# B&R Automation Studio project A2019059_Linka_Power_CP (part 41)

#### Main.st - Init, cyclic, exit code
```iecst
PROGRAM _INIT
    Triger_0:= FALSE;
    Triger_1:= FALSE;

    P4_FunkcnyTestA.STAV.Tester_ON:= TRUE;
    P4_FunkcnyTestA.OUT.HorneKontakty_ZASUN_YV177:= TRUE;
END_PROGRAM

PROGRAM _CYCLIC

	//Volanie podprogramov//
    OvlCentrovacky;
    IOLinkKomunikacia;
    OvlHornychKontaktov;
    OvlSpodnychKontaktov;
    OvlTestera;

    //Volanie funkcie SequenceControl//
    SequenceControl(SC:= SC_P4_FunkcnyTestA);

    //Príznak funkčný test A východzia pozícia//
    IF P4_FunkcnyTestA.IN.Centrovanie_ZASUNUTE_MS27 AND P4_FunkcnyTestA.IN.HorneKontakty_ZASUNUTE_MS23 AND P4_FunkcnyTestA.IN.SpodneKontakty_ZASUNUTE_MS31 THEN
        P4_FunkcnyTestA_VychodziaPozicia:= TRUE;
    ELSE
        P4_FunkcnyTestA_VychodziaPozicia:= FALSE;
    END_IF

    //Reset sekcie //
    IF NOT Safety.STAV.P4_ZonaBunky_AKTIVNA THEN
        SC_P4_FunkcnyTestA.Step:= 0;
    ELSIF P4_FunkcnyTestA.Reset THEN
        SC_P4_FunkcnyTestA.Step:= 0;
        P4_FunkcnyTestA.Reset:= FALSE;
    END_IF

    //Porucha stanice//
    IF P4_PoruchaST1 AND NOT Triger_0 THEN
        Triger_0:= TRUE;
        SC_P4_FunkcnyTestA.Step:= 0;
    END_IF

    IF NOT P4_PoruchaST1 THEN
        Triger_0:= FALSE;
    END_IF

    //Čas testovania//
    CasTestovania.PT:= T#5M;
    CasTestovania();
    NameranyCasTestovania;

    CASE SC_P4_FunkcnyTestA.Step OF

        0:
            SC_P4_FunkcnyTestA.StepName:='0 - Nulovanie';
            SC_OvlCentrovacky.Step:= 0;
            SC_OvlHornychKontaktov.Step:= 0;
            SC_OvlSpodnychKontaktov.Step:= 0;
            P4_FunkcnyTestA.Automat:= FALSE;
            P4_FunkcnyTestA.KoniecCyklu:= FALSE;
            P4_FunkcnyTestA.Manual:= FALSE;
            P4_FunkcnyTestA.STAV.PoINIT:= FALSE;
            P4_FunkcnyTestA.OUT.KontaktyTestera_VYSUN_YV171:= FALSE;
            P4_FunkcnyTestA.OUT.OdpruzenieKontaktov_VYPNI_YV180:= TRUE;
            P4_FunkcnyTestA.OUT.OdpruzenieKontaktov_ZAPNI_YV179:= FALSE;
            P4_FunkcnyTestA.OUT.ZasunStoper_YV163:= FALSE;
            PrecitaneCisloPaletky:= '';
            FV_Test_START:= FALSE;
            FV_Test_UKONCENY:= FALSE;
            Taktime_FunkcnyTestA.CMD.START_Merania_1:= FALSE;
            Taktime_FunkcnyTestA.CMD.START_Merania_2:= FALSE;
            PaletkaPrechadza:= FALSE;
            P4_FunkcnyTestA.STAV.PrebiehaVyvezeniePaletky:= FALSE;
            P4_FunkcnyTestA_ZATVOR:= FALSE;
            P4_FunkcnyTestA_OTVOR:= FALSE;
            TestovaciKus:= FALSE;
            Revork:= FALSE;
            CasTestovania.IN:= FALSE;
            P4_FunkcnyTestA.RR_TestovanieFunkcnehoTestu:= FALSE;
            P4_FunkcnyTestA.RR_VysunKontaktyTestera:= FALSE;
            P4_FunkcnyTestA.RR_ZapniOdpruzenieKontaktov:= FALSE;
            P4_FunkcnyTestA.RR_OtvorTester:= FALSE;
            P4_FunkcnyTestA.RR_ZatvorTester:= FALSE;
            PocetOpakovaniTestu:= 0;
            OpakovanyTest:= FALSE;

            IF Safety.STAV.P4_ZonaBunky_AKTIVNA AND NOT P4_Pracovisko.STAV.PORUCHA AND P4_Pracovisko.IN.PrivodVzduchu_SnimacTlaku_S15 THEN
                SC_P4_FunkcnyTestA.ResetStep:= TRUE;
                SC_P4_FunkcnyTestA.Step:= 1;
            END_IF

        1:
            SC_P4_FunkcnyTestA.StepName:='1 - Cakam na spustenie vyroby';
            P4_FunkcnyTestA.KoniecCyklu:= FALSE;
            IF P4_FunkcnyTestA.Automat THEN
                SC_P4_FunkcnyTestA.Step:= 2;
            ELSIF P4_FunkcnyTestA.Manual THEN
                SC_P4_FunkcnyTestA.Step:= 700;
            ELSIF P4_FunkcnyTestA_ZATVOR THEN
                SC_P4_FunkcnyTestA.Step:= 720;
            ELSIF P4_FunkcnyTestA_OTVOR THEN
                SC_P4_FunkcnyTestA.Step:= 750;
            END_IF

            //********************************************************Inicializácia****************************************************************************//

        2:
            SC_P4_FunkcnyTestA.StepName:='2 - Inicializacia - cakam na spustenie inicializacie';
            SC_P4_FunkcnyTestA.IdleTime.PT:= T#2s;
            SC_P4_FunkcnyTestA.AlarmTime.PT:= T#5s;

            SC_P4_FunkcnyTestA.IdleTime.IN:= TRUE;

            IF SC_P4_FunkcnyTestA.IdleTime.Q THEN
                SC_P4_FunkcnyTestA.ResetStep:= TRUE;
                SC_P4_FunkcnyTestA.Step:= 3;
            END_IF

        3:
            SC_P4_FunkcnyTestA.StepName:='3 - Inicializacia - zasunutie hornych kontaktov';
            SC_P4_FunkcnyTestA.IdleTime.PT:= T#2s;
            SC_P4_FunkcnyTestA.AlarmTime.PT:= T#5s;

            IF NOT SC_P4_FunkcnyTestA.Switch1 THEN
                HorneKontakty_ZASUN:= TRUE;
                SC_P4_FunkcnyTestA.Switch1:= TRUE;
            END_IF

            IF P4_FunkcnyTestA.IN.HorneKontakty_ZASUNUTE_MS23 THEN
                SC_P4_FunkcnyTestA.ResetStep:= TRUE;
                SC_P4_FunkcnyTestA.Step:= 5;
            END_IF

        5:
            SC_P4_FunkcnyTestA.StepName:='5 - Inicializacia - zasunutie spodnych kontaktov';
            SC_P4_FunkcnyTestA.IdleTime.PT:= T#2s;
            SC_P4_FunkcnyTestA.AlarmTime.PT:= T#5s;

            IF NOT SC_P4_FunkcnyTestA.Switch1 THEN
                SpodneKontakty_ZASUN:= TRUE;
                SC_P4_FunkcnyTestA.Switch1:= TRUE;
            END_IF

            IF P4_FunkcnyTestA.IN.SpodneKontakty_ZASUNUTE_MS31 THEN
                SC_P4_FunkcnyTestA.ResetStep:= TRUE;
                SC_P4_FunkcnyTestA.Step:= 8;
            END_IF

        8:
            SC_P4_FunkcnyTestA.StepName:='8 - Inicializacia - zasunutie centrovacky';
            SC_P4_FunkcnyTestA.IdleTime.PT:= T#4s;
            SC_P4_FunkcnyTestA.AlarmTime.PT:= T#5s;

            IF NOT SC_P4_FunkcnyTestA.Switch1 THEN
                Centrovacku_ZASUN:= TRUE;
                SC_P4_FunkcnyTestA.Switch1:= TRUE;
            END_IF

            IF P4_FunkcnyTestA.IN.Centrovanie_ZASUNUTE_MS27 AND P4_Dopravniky.STAV.PoINIT THEN
                SC_P4_FunkcnyTestA.ResetStep:= TRUE;
                SC_P4_FunkcnyTestA.Step:= 10;
            END_IF

        10:
            SC_P4_FunkcnyTestA.StepName:='10 - Inicializacia - kontrola kontaktov funkcneho testu';
            SC_P4_FunkcnyTestA.IdleTime.PT:= T#4s;
            SC_P4_FunkcnyTestA.AlarmTime.PT:= T#5s;

            IF Linka.PAR.ZvolenyModel = '4F' AND P4_FunkcnyTestA.IN.TypSpodnychKontaktov_4F THEN
                SC_P4_FunkcnyTestA.ResetStep:= TRUE;
                SC_P4_FunkcnyTestA.Step:= 13;
            ELSIF Linka.PAR.ZvolenyModel = '5F' AND P4_FunkcnyTestA.IN.TypSpodnychKontaktov_5F_5H THEN
                SC_P4_FunkcnyTestA.ResetStep:= TRUE;
                SC_P4_FunkcnyTestA.Step:= 13;
            ELSIF Linka.PAR.ZvolenyModel = '5H'AND P4_FunkcnyTestA.IN.TypSpodnychKontaktov_5F_5H THEN
                SC_P4_FunkcnyTestA.ResetStep:= TRUE;
                SC_P4_FunkcnyTestA.Step:= 13;
            ELSE
                P34_Alarmy[437]:= TRUE;
                P4_PoruchaST1:= TRUE;
            END_IF

        13:
            SC_P4_FunkcnyTestA.StepName:='13 - Inicializacia - hladanie paletky';
            SC_P4_FunkcnyTestA.IdleTime.PT:= T#5s;
            SC_P4_FunkcnyTestA.AlarmTime.PT:= T#5s;
            SC_P4_FunkcnyTestA.IdleTime.IN:= TRUE;

            IF P4_FunkcnyTestA.IN.PritomnostPaletky_S10 THEN
                P3_LeakageTestB.STAV.PrebiehaVyvezeniePaletky:= FALSE;
                SC_P4_FunkcnyTestA.ResetStep:= TRUE;
                SC_P4_FunkcnyTestA.Step:= 20;
            ELSIF SC_P4_FunkcnyTestA.IdleTime.Q THEN
                P4_FunkcnyTestA.STAV.PoINIT:= TRUE;
                SC_P4_FunkcnyTestA.ResetStep:= TRUE;
                SC_P4_FunkcnyTestA.Step:= 100;
            END_IF

        20:
            SC_P4_FunkcnyTestA.StepName:='20 - Inicializacia - precitanie cisla paletky';
            SC_P4_FunkcnyTestA.IdleTime.PT:= T#200ms;
            SC_P4_FunkcnyTestA.AlarmTime.PT:= T#5s;
            SC_P4_FunkcnyTestA.IdleTime.IN:= TRUE;

            IF SC_P4_FunkcnyTestA.IdleTime.Q THEN
                PrecitaneCisloPaletky:= USINT_TO_STRING(P4_FunkcnyTestA.IN.PrecitaneCisloPaletky_S10);
                i:= 0;
                SC_P4_FunkcnyTestA.ResetStep:= TRUE;
                SC_P4_FunkcnyTestA.Step:= 23;
            END_IF

        23:
            SC_P4_FunkcnyTestA.StepName:='23 - Inicializacia - priradenie indexu paletky na zaklade precitanej hodnoty';
            SC_P4_FunkcnyTestA.IdleTime.PT:= T#200ms;
            SC_P4_FunkcnyTestA.AlarmTime.PT:= T#5s;

            IF PrecitaneCisloPaletky = '171' THEN
                i:= 1;
            ELSIF PrecitaneCisloPaletky = '164' THEN
                i:= 2;
            ELSIF PrecitaneCisloPaletky = '181' THEN
                i:= 3;
            ELSIF PrecitaneCisloPaletky = '168' THEN
                i:= 4;
            ELSIF PrecitaneCisloPaletky = '140' THEN
                i:= 5;
            ELSIF PrecitaneCisloPaletky = '110' THEN
                i:= 6;
            ELSIF PrecitaneCisloPaletky = '156' THEN
                i:= 7;
            ELSIF PrecitaneCisloPaletky = '127' THEN
                i:= 8;
            ELSIF PrecitaneCisloPaletky = '139' THEN
                i:= 9;
            ELSIF PrecitaneCisloPaletky = '131' THEN
                i:= 10;
            ELSIF PrecitaneCisloPaletky = '178' THEN
                i:= 11;
            ELSIF PrecitaneCisloPaletky = '206' THEN
                i:= 12;
            ELSIF PrecitaneCisloPaletky = '119' THEN
                i:= 13;
            ELSIF PrecitaneCisloPaletky = '163' THEN
                i:= 14;
            ELSIF PrecitaneCisloPaletky = '128' THEN
                i:= 15;
            ELSIF PrecitaneCisloPaletky = '175' THEN
                i:= 16;
            ELSIF PrecitaneCisloPaletky = '138' THEN
                i:= 17;
            ELSE
                P34_Alarmy[427]:= TRUE;
                P4_PoruchaST1:= TRUE;
            END_IF

            IF i<> 0 THEN
                Paletka[i].PAR.CisloPaletky:= USINT_TO_STRING(i);
                PrecitaneCisloPaletky:= '';
                SC_P4_FunkcnyTestA.ResetStep:= TRUE;
                SC_P4_FunkcnyTestA.Step:= 30;
            END_IF

        30:
            SC_P4_FunkcnyTestA.StepName:='30 - Inicializacia - kontrola stavu paletky';
            SC_P4_FunkcnyTestA.IdleTime.PT:= T#200ms;
            SC_P4_FunkcnyTestA.AlarmTime.PT:= T#5s;

            IF Paletka[i].PAR.TestovaciKus AND Paletka[i].PAR.CisloTestovacejStanice = 'ST_FT1,FT2' THEN
                IF P4_FunkcnyTestA.STAV.Tester_ON THEN
                    TestovaciKus:= TRUE;
                    P4_FunkcnyTestA.STAV.PoINIT:= TRUE;
                    SC_P4_FunkcnyTestA.ResetStep:= TRUE;
                    SC_P4_FunkcnyTestA.Step:= 118;
                ELSE
                    P4_FunkcnyTestA.STAV.PoINIT:= TRUE;
                    SC_P4_FunkcnyTestA.ResetStep:= TRUE;
                    SC_P4_FunkcnyTestA.Step:= 560;
                END_IF
            ELSIF Paletka[i].PAR.TestovaciKus AND Paletka[i].PAR.CisloTestovacejStanice <> 'ST_FT1,FT2' THEN
                P4_FunkcnyTestA.STAV.PoINIT:= TRUE;
                SC_P4_FunkcnyTestA.ResetStep:= TRUE;
                SC_P4_FunkcnyTestA.Step:= 560;
            ELSIF Paletka[i].PAR.RevorkovyKus AND Paletka[i].PAR.CisloRevorkovejStanice = 'ST_FT1,FT2' THEN
                IF P4_FunkcnyTestA.STAV.Tester_ON THEN
                    Revork:= TRUE;
                    P4_FunkcnyTestA.STAV.PoINIT:= TRUE;
                    SC_P4_FunkcnyTestA.ResetStep:= TRUE;
                    SC_P4_FunkcnyTestA.Step:= 105;
                ELSE
                    P4_FunkcnyTestA.STAV.PoINIT:= TRUE;
                    SC_P4_FunkcnyTestA.ResetStep:= TRUE;
                    SC_P4_FunkcnyTestA.Step:= 560;
                END_IF
            ELSIF Paletka[i].PAR.RevorkovyKus AND Paletka[i].PAR.CisloRevorkovejStanice <> 'ST_FT1,FT2' THEN
                Revork:= FALSE;
                P4_FunkcnyTestA.STAV.PoINIT:= TRUE;
                SC_P4_FunkcnyTestA.ResetStep:= TRUE;
                SC_P4_FunkcnyTestA.Step:= 560;
            ELSIF Paletka[i].PAR.StavPaletky = 'OK' THEN
                SC_P4_FunkcnyTestA.ResetStep:= TRUE;
                SC_P4_FunkcnyTestA.Step:= 33;
            ELSIF Paletka[i].PAR.StavPaletky = 'NG' THEN
                P4_FunkcnyTestA.STAV.PoINIT:= TRUE;
                SC_P4_FunkcnyTestA.ResetStep:= TRUE;
                SC_P4_FunkcnyTestA.Step:= 560;
            END_IF

        33:
            SC_P4_FunkcnyTestA.StepName:='33 - Inicializacia - kontrola ukoncenia testu';
            SC_P4_FunkcnyTestA.IdleTime.PT:= T#200ms;
            SC_P4_FunkcnyTestA.AlarmTime.PT:= T#5s;

            IF Paletka[i].VnutornyStav.FunkcnyTest_Ukonceny THEN
                P4_FunkcnyTestA.STAV.PoINIT:= TRUE;
                SC_P4_FunkcnyTestA.ResetStep:= TRUE;
                SC_P4_FunkcnyTestA.Step:= 560;
            ELSE
                P4_FunkcnyTestA.STAV.PoINIT:= TRUE;
                SC_P4_FunkcnyTestA.ResetStep:= TRUE;
                SC_P4_FunkcnyTestA.Step:= 100;
            END_IF

            //********************************************************Automatický režim****************************************************************************//

        100:
            SC_P4_FunkcnyTestA.StepName:='100 - Automaticky Rezim - cakam na príchod paletky na stoper';
            SC_P4_FunkcnyTestA.IdleTime.PT:= T#200ms;
            SC_P4_FunkcnyTestA.AlarmTime.PT:= T#5s;

            IF P4_FunkcnyTestA.IN.PritomnostPaletky_S10 THEN
                P3_LeakageTestB.STAV.PrebiehaVyvezeniePaletky:= FALSE;
            END_IF

            SC_P4_FunkcnyTestA.IdleTime.IN:= P4_FunkcnyTestA.IN.PritomnostPaletky_S10;

            IF EDGEPOS(P4_FunkcnyTestA.IN.PritomnostPaletky_S10)THEN
                IF NOT Taktime_FunkcnyTestA.CMD.START_Merania_1 THEN
                    Taktime_FunkcnyTestA.CMD.START_Merania_1:= TRUE;
                ELSE
                    Taktime_FunkcnyTestA.CMD.ZAPIS_Hodnot_1:= TRUE;
                END_IF
            END_IF

            IF P4_FunkcnyTestA.KoniecCyklu THEN
                SC_P4_FunkcnyTestA.ResetStep:= TRUE;
                SC_P4_FunkcnyTestA.Step:= 0;
            ELSIF SC_P4_FunkcnyTestA.IdleTime.Q THEN
                SC_P4_FunkcnyTestA.ResetStep:= TRUE;
                SC_P4_FunkcnyTestA.Step:= 101;
            END_IF

        101:
            SC_P4_FunkcnyTestA.StepName:='101 - Automaticky Rezim - precitanie cisla paletky';
            SC_P4_FunkcnyTestA.IdleTime.PT:= T#500ms;
            SC_P4_FunkcnyTestA.AlarmTime.PT:= T#5s;
            SC_P4_FunkcnyTestA.IdleTime.IN:= TRUE;

            PrecitaneCisloPaletky:= USINT_TO_STRING(P4_FunkcnyTestA.IN.PrecitaneCisloPaletky_S10);
            i:= 0;
            SC_P4_FunkcnyTestA.ResetStep:= TRUE;
            SC_P4_FunkcnyTestA.Step:= 102;

        102:
            SC_P4_FunkcnyTestA.StepName:='102 - Automaticky Rezim - priradenie indexu paletky na zaklade precitanej hodnoty';
            SC_P4_FunkcnyTestA.IdleTime.PT:= T#200ms;
            SC_P4_FunkcnyTestA.AlarmTime.PT:= T#5s;

            IF PrecitaneCisloPaletky = '171' THEN
                i:= 1;
            ELSIF PrecitaneCisloPaletky = '164' THEN
                i:= 2;
            ELSIF PrecitaneCisloPaletky = '181' THEN
                i:= 3;
            ELSIF PrecitaneCisloPaletky = '168' THEN
                i:= 4;
            ELSIF PrecitaneCisloPaletky = '140' THEN
                i:= 5;
            ELSIF PrecitaneCisloPaletky = '110' THEN
                i:= 6;
            ELSIF PrecitaneCisloPaletky = '156' THEN
                i:= 7;
            ELSIF PrecitaneCisloPaletky = '127' THEN
                i:= 8;
            ELSIF PrecitaneCisloPaletky = '139' THEN
                i:= 9;
            ELSIF PrecitaneCisloPaletky = '131' THEN
                i:= 10;
            ELSIF PrecitaneCisloPaletky = '178' THEN
                i:= 11;
            ELSIF PrecitaneCisloPaletky = '206' THEN
                i:= 12;
            ELSIF PrecitaneCisloPaletky = '119' THEN
                i:= 13;
            ELSIF PrecitaneCisloPaletky = '163' THEN
                i:= 14;
            ELSIF PrecitaneCisloPaletky = '128' THEN
                i:= 15;
            ELSIF PrecitaneCisloPaletky = '175' THEN
                i:= 16;
            ELSIF PrecitaneCisloPaletky = '138' THEN
                i:= 17;
            ELSE
                P34_Alarmy[427]:= TRUE;
                P4_PoruchaST1:= TRUE;
            END_IF

            IF i<> 0 THEN
                Paletka[i].PAR.CisloPaletky:= USINT_TO_STRING(i);
                PrecitaneCisloPaletky:= '';
                SC_P4_FunkcnyTestA.ResetStep:= TRUE;
                SC_P4_FunkcnyTestA.Step:= 103;
            END_IF

        103:
            SC_P4_FunkcnyTestA.StepName:='108 - Automaticky Rezim - kontrola stavu paletky';
            SC_P4_FunkcnyTestA.IdleTime.PT:= T#200ms;
            SC_P4_FunkcnyTestA.AlarmTime.PT:= T#5s;

            IF Paletka[i].PAR.TestovaciKus AND Paletka[i].PAR.CisloTestovacejStanice = 'ST_FT1,FT2' THEN
                IF P4_FunkcnyTestA.STAV.Tester_ON THEN
                    TestovaciKus:= TRUE;
                    SC_P4_FunkcnyTestA.ResetStep:= TRUE;
                    SC_P4_FunkcnyTestA.Step:= 118;
                ELSE
                    SC_P4_FunkcnyTestA.ResetStep:= TRUE;
                    SC_P4_FunkcnyTestA.Step:= 560;
                END_IF
            ELSIF Paletka[i].PAR.TestovaciKus AND Paletka[i].PAR.CisloTestovacejStanice <> 'ST_FT1,FT2' THEN
                SC_P4_FunkcnyTestA.ResetStep:= TRUE;
                SC_P4_FunkcnyTestA.Step:= 560;
            ELSIF Paletka[i].PAR.RevorkovyKus AND Paletka[i].PAR.CisloRevorkovejStanice = 'ST_FT1,FT2' THEN
                IF P4_FunkcnyTestA.STAV.Tester_ON THEN
                    Revork:= TRUE;
                    SC_P4_FunkcnyTestA.ResetStep:= TRUE;
                    SC_P4_FunkcnyTestA.Step:= 105;
                ELSE
                    SC_P4_FunkcnyTestA.ResetStep:= TRUE;
                    SC_P4_FunkcnyTestA.Step:= 560;
                END_IF
            ELSIF Paletka[i].PAR.RevorkovyKus AND Paletka[i].PAR.CisloRevorkovejStanice <> 'ST_FT1,FT2' THEN
                Revork:= FALSE;
                SC_P4_FunkcnyTestA.ResetStep:= TRUE;
                SC_P4_FunkcnyTestA.Step:= 560;
            ELSIF Paletka[i].PAR.StavPaletky = 'OK' AND P4_FunkcnyTestA.STAV.Tester_ON THEN
                SC_P4_FunkcnyTestA.ResetStep:= TRUE;
                SC_P4_FunkcnyTestA.Step:= 105;
            ELSIF Paletka[i].PAR.StavPaletky = 'OK' AND NOT P4_FunkcnyTestA.STAV.Tester_ON THEN
                SC_P4_FunkcnyTestA.ResetStep:= TRUE;
                SC_P4_FunkcnyTestA.Step:= 560;
            ELSIF Paletka[i].PAR.StavPaletky = 'NG' THEN
                SC_P4_FunkcnyTestA.ResetStep:= TRUE;
                SC_P4_FunkcnyTestA.Step:= 560;
            END_IF

        105:
            SC_P4_FunkcnyTestA.StepName:='105 - Automaticky Rezim - kontrola zapnutia testovacej stanice B';
            SC_P4_FunkcnyTestA.IdleTime.PT:= T#200ms;
            SC_P4_FunkcnyTestA.AlarmTime.PT:= T#5s;

            IF P4_FunkcnyTestB.STAV.Tester_ON THEN
                SC_P4_FunkcnyTestA.ResetStep:= TRUE;
                SC_P4_FunkcnyTestA.Step:= 107;
            ELSE
                SC_P4_FunkcnyTestA.ResetStep:= TRUE;
                SC_P4_FunkcnyTestA.Step:= 118;
            END_IF

        107:
            SC_P4_FunkcnyTestA.StepName:='107 - Automaticky Rezim - kontrola paletky v testovacej stanici B';
            SC_P4_FunkcnyTestA.IdleTime.PT:= T#1s;
            SC_P4_FunkcnyTestA.AlarmTime.PT:= T#5s;
            SC_P4_FunkcnyTestA.IdleTime.IN:= TRUE;

            IF P4_FunkcnyTestA.KoniecCyklu THEN
                SC_P4_FunkcnyTestA.ResetStep:= TRUE;
                SC_P4_FunkcnyTestA.Step:= 118;
            ELSIF SC_P4_FunkcnyTestB.Step = 100 AND NOT P4_FunkcnyTestB.IN.PritomnostPaletky_S11 THEN
                SC_P4_FunkcnyTestA.ResetStep:= TRUE;
                SC_P4_FunkcnyTestA.Step:= 560;
            ELSIF SC_P4_FunkcnyTestB.Step = 110 AND P4_FunkcnyTestB.IN.PritomnostPaletky_S11 THEN
                SC_P4_FunkcnyTestA.ResetStep:= TRUE;
                SC_P4_FunkcnyTestA.Step:= 110;
            END_IF

        110:
            SC_P4_FunkcnyTestA.StepName:='110 - Automaticky Rezim - cakam na spustenie testovania';
            SC_P4_FunkcnyTestA.IdleTime.PT:= T#200ms;
            SC_P4_FunkcnyTestA.AlarmTime.PT:= T#5s;

            IF P4_FunkcnyTestB.OUT.KOM_StanicaA_StartTestovania THEN
                P4_FunkcnyTestB.OUT.KOM_StanicaA_StartTestovania:= FALSE;
                SC_P4_FunkcnyTestA.ResetStep:= TRUE;
                SC_P4_FunkcnyTestA.Step:= 118;
            END_IF

        118:
            SC_P4_FunkcnyTestA.StepName:='118 - Automaticky Rezim - zacentrovanie paletky';
            SC_P4_FunkcnyTestA.IdleTime.PT:= T#200ms;
            SC_P4_FunkcnyTestA.AlarmTime.PT:= T#5s;

            IF NOT SC_P4_FunkcnyTestA.Switch1 THEN
                Centrovacku_VYSUN:= TRUE;
                SC_P4_FunkcnyTestA.Switch1:= TRUE;
            END_IF

            IF P4_FunkcnyTestA.IN.Centrovanie_VYSUNUTE_MS29 THEN
                SC_P4_FunkcnyTestA.ResetStep:= TRUE;
                SC_P4_FunkcnyTestA.Step:= 120;
            END_IF

        120:
            SC_P4_FunkcnyTestA.StepName:='120 - Automaticky Rezim - zapnutie pruzenia vrchnych kontaktov';
            SC_P4_FunkcnyTestA.IdleTime.PT:= T#200ms;
            SC_P4_FunkcnyTestA.AlarmTime.PT:= T#5s;

            IF NOT SC_P4_FunkcnyTestA.Switch1 THEN
                P4_FunkcnyTestA.OUT.OdpruzenieKontaktov_VYPNI_YV180:= FALSE;
                P4_FunkcnyTestA.OUT.OdpruzenieKontaktov_ZAPNI_YV179:= TRUE;
                SC_P4_FunkcnyTestA.IdleTime.IN:= TRUE;
                SC_P4_FunkcnyTestA.Switch1:= TRUE;
            END_IF

            IF SC_P4_FunkcnyTestA.IdleTime.Q THEN
                SC_P4_FunkcnyTestA.ResetStep:= TRUE;
                SC_P4_FunkcnyTestA.Step:= 123;
            END_IF

        123:
            SC_P4_FunkcnyTestA.StepName:='123 - Automaticky Rezim - vysunutie hornych kontaktov';
            SC_P4_FunkcnyTestA.IdleTime.PT:= T#200ms;
            SC_P4_FunkcnyTestA.AlarmTime.PT:= T#5s;

            IF NOT SC_P4_FunkcnyTestA.Switch1 THEN
                HorneKontakty_VYSUN:= TRUE;
                SC_P4_FunkcnyTestA.Switch1:= TRUE;
            END_IF

            IF P4_FunkcnyTestA.IN.HorneKontakty_VYSUNUTE_MS25 THEN
                SC_P4_FunkcnyTestA.ResetStep:= TRUE;
                SC_P4_FunkcnyTestA.Step:= 125;
            END_IF

        125:
            SC_P4_FunkcnyTestA.StepName:='125 - Automaticky Rezim - vysunutie spodnych kontaktov';
            SC_P4_FunkcnyTestA.IdleTime.PT:= T#200ms;
            SC_P4_FunkcnyTestA.AlarmTime.PT:= T#5s;

            IF NOT SC_P4_FunkcnyTestA.Switch1 THEN
                SpodneKontakty_VYSUN:= TRUE;
                SC_P4_FunkcnyTestA.Switch1:= TRUE;
            END_IF

            IF P4_FunkcnyTestA.IN.SpodneKontakty_VYSUNUTE_MS33 THEN
                SC_P4_FunkcnyTestA.ResetStep:= TRUE;
                SC_P4_FunkcnyTestA.Step:= 127;
            END_IF

        127:
            SC_P4_FunkcnyTestA.StepName:='127 - Automaticky Rezim - pritlacenie kontaktov';
            SC_P4_FunkcnyTestA.IdleTime.PT:= T#200ms;
            SC_P4_FunkcnyTestA.AlarmTime.PT:= T#5s;

            IF Linka.PAR.ZvolenyModel = '4F' THEN
                P4_FunkcnyTestA.OUT.KontaktyTestera_VYSUN_YV171:= TRUE;
                SC_P4_FunkcnyTestA.IdleTime.IN:= TRUE;
            ELSIF Linka.PAR.ZvolenyModel = '5F' THEN
                P4_FunkcnyTestA.OUT.KontaktyTestera_VYSUN_YV171:= TRUE;
                SC_P4_FunkcnyTestA.IdleTime.IN:= TRUE;
            ELSIF Linka.PAR.ZvolenyModel = '5H' THEN
                SC_P4_FunkcnyTestA.ResetStep:= TRUE;
                SC_P4_FunkcnyTestA.Step:= 130;
            END_IF

            IF SC_P4_FunkcnyTestA.IdleTime.Q THEN
                SC_P4_FunkcnyTestA.ResetStep:= TRUE;
                SC_P4_FunkcnyTestA.Step:= 130;
            END_IF

        130:
            SC_P4_FunkcnyTestA.StepName:='130 - Automaticky Rezim - spustenie testovania';
            SC_P4_FunkcnyTestA.IdleTime.PT:= T#5s;
            SC_P4_FunkcnyTestA.AlarmTime.PT:= T#5s;

            IF NOT SC_P4_FunkcnyTestA.Switch1 THEN
                FV_Test_UKONCENY:= FALSE;
                FV_Test_START:= TRUE;
                CasTestovania.IN:= TRUE;
                SC_P4_FunkcnyTestA.Switch1:= TRUE;
            END_IF

            IF FV_Test_START AND FV_Test_UKONCENY THEN
                FV_Test_START:= FALSE;
                SC_P4_FunkcnyTestA.ResetStep:= TRUE;
                SC_P4_FunkcnyTestA.Step:= 140;
            END_IF

        140:
            SC_P4_FunkcnyTestA.StepName:='140 - Automaticky Rezim - vyhodnotenie testovania';
            SC_P4_FunkcnyTestA.IdleTime.PT:= T#200ms;
            SC_P4_FunkcnyTestA.AlarmTime.PT:= T#5s;

            IF P4_FunkcnyTestA.STAV.Vysledok_FV_Testu = 'OK' THEN
                Paletka[i].PAR.StavPowerCP:= 'PASS';
                Paletka[i].PAR.StavPaletky:= 'OK';
                Paletka[i].VnutornyStav.FunkcnyTest_Ukonceny:= TRUE;
                SC_P4_FunkcnyTestA.ResetStep:= TRUE;
                SC_P4_FunkcnyTestA.Step:= 145;
            ELSIF P4_FunkcnyTestA.STAV.Vysledok_FV_Testu = 'NG' THEN
                IF NOT Revork THEN
                    OpakovanyTest:= TRUE;
                END_IF
                Paletka[i].PAR.StavPowerCP:= 'FAIL';
                Paletka[i].PAR.StavPaletky:= 'NG';
                SC_P4_FunkcnyTestA.ResetStep:= TRUE;
                SC_P4_FunkcnyTestA.Step:= 145;
            END_IF

        145:
            SC_P4_FunkcnyTestA.StepName:='127 - Automaticky Rezim - vypnutie pritlacenie kontaktov';
            SC_P4_FunkcnyTestA.IdleTime.PT:= T#200ms;
            SC_P4_FunkcnyTestA.AlarmTime.PT:= T#5s;

            P4_FunkcnyTestA.OUT.KontaktyTestera_VYSUN_YV171:= FALSE;
            SC_P4_FunkcnyTestA.ResetStep:= TRUE;
            SC_P4_FunkcnyTestA.Step:= 148;

        148:
            SC_P4_FunkcnyTestA.StepName:='148 - Automaticky Rezim - zasunutie spodnych kontaktov';
            SC_P4_FunkcnyTestA.IdleTime.PT:= T#200ms;
            SC_P4_FunkcnyTestA.AlarmTime.PT:= T#5s;

            IF NOT SC_P4_FunkcnyTestA.Switch1 THEN
                SpodneKontakty_ZASUN:= TRUE;
                SC_P4_FunkcnyTestA.Switch1:= TRUE;
            END_IF

            IF P4_FunkcnyTestA.IN.SpodneKontakty_ZASUNUTE_MS31 THEN
                SC_P4_FunkcnyTestA.ResetStep:= TRUE;
                SC_P4_FunkcnyTestA.Step:= 150;
            END_IF

        150:
            SC_P4_FunkcnyTestA.StepName:='150 - Automaticky Rezim - zasunutie hornych kontaktov';
            SC_P4_FunkcnyTestA.IdleTime.PT:= T#200ms;
            SC_P4_FunkcnyTestA.AlarmTime.PT:= T#5s;

            IF NOT SC_P4_FunkcnyTestA.Switch1 THEN
                HorneKontakty_ZASUN:= TRUE;
                SC_P4_FunkcnyTestA.Switch1:= TRUE;
            END_IF

            IF P4_FunkcnyTestA.IN.HorneKontakty_ZASUNUTE_MS23 THEN
                SC_P4_FunkcnyTestA.ResetStep:= TRUE;
                SC_P4_FunkcnyTestA.Step:= 153;
            END_IF

        153:
            SC_P4_FunkcnyTestA.StepName:='153 - Automaticky Rezim - vypnutie pruzenia vrchnych kontaktov';
            SC_P4_FunkcnyTestA.IdleTime.PT:= T#200ms;
            SC_P4_FunkcnyTestA.AlarmTime.PT:= T#5s;

            IF NOT SC_P4_FunkcnyTestA.Switch1 THEN
                P4_FunkcnyTestA.OUT.OdpruzenieKontaktov_ZAPNI_YV179:= FALSE;
                P4_FunkcnyTestA.OUT.OdpruzenieKontaktov_VYPNI_YV180:= TRUE;
                SC_P4_FunkcnyTestA.IdleTime.IN:= TRUE;
                SC_P4_FunkcnyTestA.Switch1:= TRUE;
            END_IF

            IF SC_P4_FunkcnyTestA.IdleTime.Q THEN
                SC_P4_FunkcnyTestA.ResetStep:= TRUE;
                SC_P4_FunkcnyTestA.Step:= 545;
            END_IF

            //Odcentrovanie paletky//

        545:
            SC_P4_FunkcnyTestA.StepName:='545 - Automaticky Rezim - odcentrovanie paletky';
            SC_P4_FunkcnyTestA.IdleTime.PT:= T#200ms;
            SC_P4_FunkcnyTestA.AlarmTime.PT:= T#5s;

            IF NOT SC_P4_FunkcnyTestA.Switch1 THEN
                Centrovacku_ZASUN:= TRUE;
                SC_P4_FunkcnyTestA.Switch1:= TRUE;
            END_IF

            IF P4_FunkcnyTestA.IN.Centrovanie_ZASUNUTE_MS27 THEN
                SC_P4_FunkcnyTestA.ResetStep:= TRUE;
                SC_P4_FunkcnyTestA.Step:= 554;
            END_IF

        554:
            SC_P4_FunkcnyTestA.StepName:='554 - Automaticky Rezim - kontrola poctu testovani';
            SC_P4_FunkcnyTestA.IdleTime.PT:= T#1s;
            SC_P4_FunkcnyTestA.AlarmTime.PT:= T#5s;
            SC_P4_FunkcnyTestA.IdleTime.IN:= TRUE;

            IF NOT SC_P4_FunkcnyTestA.Switch1 THEN
                PocetOpakovaniTestu:= PocetOpakovaniTestu + 1;
                SC_P4_FunkcnyTestA.Switch1:= TRUE;
            END_IF

            IF OpakovanyTest AND PocetOpakovaniTestu < 2 AND SC_P4_FunkcnyTestA.IdleTime.Q AND NOT TestovaciKus THEN
                OpakovanyTest:= FALSE;
                SC_P4_FunkcnyTestA.ResetStep:= TRUE;
                SC_P4_FunkcnyTestA.Step:= 118;
            ELSIF OpakovanyTest AND PocetOpakovaniTestu >= 2 AND NOT TestovaciKus THEN
                Paletka[i].VnutornyStav.FunkcnyTest_Ukonceny:= TRUE;
                OpakovanyTest:= FALSE;
                PocetOpakovaniTestu:= 0;
                SC_P4_FunkcnyTestA.ResetStep:= TRUE;
                SC_P4_FunkcnyTestA.Step:= 555;
            ELSIF NOT OpakovanyTest OR TestovaciKus THEN
                SC_P4_FunkcnyTestA.ResetStep:= TRUE;
                SC_P4_FunkcnyTestA.Step:= 555;
            END_IF

        555:
            SC_P4_FunkcnyTestA.StepName:='555 - Automaticky Rezim - vyhodnotenie stavu paletky';
            SC_P4_FunkcnyTestA.IdleTime.PT:= T#200ms;
            SC_P4_FunkcnyTestA.AlarmTime.PT:= T#5s;

            IF Paletka[i].PAR.StavPaletky = 'OK' THEN
                IF Paletka[i].PAR.StavPowerCP = 'PASS' THEN
                    Paletka[i].PAR.StavPaletky:= 'OK';
                ELSIF Paletka[i].PAR.StavPowerCP = 'FAIL' THEN
                    Paletka[i].PAR.StavPaletky:= 'NG';
                END_IF
            END_IF

            SC_P4_FunkcnyTestA.ResetStep:= TRUE;
            SC_P4_FunkcnyTestA.Step:= 560;

            //Vyvezenie paletky//

        560:
            SC_P4_FunkcnyTestA.StepName:='560 - Automaticky Rezim - cakam na vyvezenie na stoper funkcneho testu B';
            SC_P4_FunkcnyTestA.IdleTime.PT:= T#200ms;
            SC_P4_FunkcnyTestA.AlarmTime.PT:= T#5s;

            IF P4_FunkcnyTestA.KoniecCyklu THEN
                SC_P4_FunkcnyTestA.ResetStep:= TRUE;
                SC_P4_FunkcnyTestA.Step:= 0;
            ELSIF ((NOT P4_FunkcnyTestB.IN.PritomnostPaletky_S11 AND SC_P4_FunkcnyTestB.Step = 100) OR (P4_FunkcnyTestB.OUT.ZasunStoper_YV164 AND SC_P4_FunkcnyTestB.Step = 561)) AND NOT P4_FunkcnyTestA.STAV.PrebiehaVyvezeniePaletky AND NOT TEST THEN
                P4_FunkcnyTestA.OUT.ZasunStoper_YV163:= TRUE;
                P4_FunkcnyTestA.STAV.PrebiehaVyvezeniePaletky:= TRUE;
                SC_P4_FunkcnyTestA.ResetStep:= TRUE;
                SC_P4_FunkcnyTestA.Step:= 561;
            END_IF

        561:
            SC_P4_FunkcnyTestA.StepName:='561 - Automaticky Rezim - ukoncenie vyvazania na stoper funkcneho testu B';
            SC_P4_FunkcnyTestA.IdleTime.PT:= T#200ms;
            SC_P4_FunkcnyTestA.AlarmTime.PT:= T#10s;

            SC_P4_FunkcnyTestA.IdleTime.IN:= NOT P4_FunkcnyTestA.IN.PritomnostPaletky_S10;
            SC_P4_FunkcnyTestA.AlarmTime.IN:= P4_FunkcnyTestA.IN.PritomnostPaletky_S10;

            IF NOT P4_FunkcnyTestA.IN.PritomnostPaletky_S10 THEN
                IF Revork THEN
                    Paletka[i].PAR.RevorkovyKus:= FALSE;
                    Paletka[i].PAR.CisloRevorkovejStanice:= '';
                    Revork:= FALSE;
                END_IF
                P4_FunkcnyTestA.OUT.ZasunStoper_YV163:= FALSE;
                TestovaciKus:= FALSE;
                OpakovanyTest:= FALSE;
                PocetOpakovaniTestu:= 0;
                Paletka[i].PAR.StavPowerCP:= '';
            END_IF

            IF SC_P4_FunkcnyTestA.IdleTime.Q AND NOT P4_FunkcnyTestA.OUT.ZasunStoper_YV163 THEN
                SC_P4_FunkcnyTestA.ResetStep:= TRUE;
                SC_P4_FunkcnyTestA.Step:= 100;
            ELSIF SC_P4_FunkcnyTestA.AlarmTime.Q THEN
                P34_Alarmy[450]:= TRUE;
                P4_Pracovisko.KoniecCyklu:= TRUE;
                SC_P4_FunkcnyTestA.ResetStep:= TRUE;
                SC_P4_FunkcnyTestA.Step:= 0;
            END_IF

            //*******************************************************Manuálny režim*******************************************************************************//
        700:
            SC_P4_FunkcnyTestA.StepName:='700 - Manualny Rezim';
            SC_P4_FunkcnyTestA.IdleTime.PT:= T#8s;
            SC_P4_FunkcnyTestA.AlarmTime.PT:= T#5s;

            //Ovládanie odpruženia kontaktov//
            IF P4_FunkcnyTestA.RR_ZapniOdpruzenieKontaktov THEN
                P4_FunkcnyTestA.OUT.OdpruzenieKontaktov_VYPNI_YV180:= FALSE;
                P4_FunkcnyTestA.OUT.OdpruzenieKontaktov_ZAPNI_YV179:= TRUE;
            ELSE
                P4_FunkcnyTestA.OUT.OdpruzenieKontaktov_ZAPNI_YV179:= FALSE;
                P4_FunkcnyTestA.OUT.OdpruzenieKontaktov_VYPNI_YV180:= TRUE;
            END_IF

            //Ovládanie vysunutia kontaktov testera//
            P4_FunkcnyTestA.OUT.KontaktyTestera_VYSUN_YV171:= P4_FunkcnyTestA.RR_VysunKontaktyTestera;

    END_CASE

                END_PROGRAM

PROGRAM _EXIT
                (* Insert code here *)

                END_PROGRAM
```

#### Variables.var - Local variables
```iecst
VAR
	SC_OvlCentrovacky : SequenceControlTyp;
	Centrovacku_VYSUN : BOOL;
	Centrovacku_ZASUN : BOOL;
	PrecitaneCisloPaletky : STRING[3];
	ServerOdpoved_StavPowerCP : STRING[5];
	i : USINT;
	SC_OvlSpodnychKontaktov : SequenceControlTyp;
	SpodneKontakty_VYSUN : BOOL;
	SpodneKontakty_ZASUN : BOOL;
	SC_OvlHornychKontaktov : SequenceControlTyp;
	HorneKontakty_VYSUN : BOOL;
	HorneKontakty_ZASUN : BOOL;
	SC_OvlTesteraFT : SequenceControlTyp;
	SKTcpClientTester_0 : SKTcpClientTester;
	dataStr : STRING[32];
	FV_Test_START : BOOL;
	FV_Test_UKONCENY : BOOL;
	TEST : BOOL;
	FV_Test_PocetDopytovTestera : USINT;
	PaletkaPrechadza : BOOL;
	TestovaciKus : BOOL;
	Revork : BOOL;
	PocetDopytovNaTester : USINT;
	CasTestovania : TON;
	NameranyCasTestovania : TIME;
	Triger_0 : BOOL;
	Triger_1 : BOOL;
	PocetOpakovaniTestu : USINT;
	OpakovanyTest : BOOL;
END_VAR
```

#### IOLinkKomunikacia.st
```iecst
ACTION IOLinkKomunikacia:

	//Snímač paletky//
	P4_FunkcnyTestA.IN.PritomnostPaletky_S10:= P4_FunkcnyTestA.PAR.SnimacPaletky_IOLinkInputs[1].0;
	P4_FunkcnyTestA.IN.PrecitaneCisloPaletky_S10:= P4_FunkcnyTestA.PAR.SnimacPaletky_IOLinkInputs[9];

END_ACTION
```

#### OvlCentrovacky.st
```iecst
ACTION OvlCentrovacky:

	//Volanie funkcie SequenceControl//
	SequenceControl(SC:= SC_OvlCentrovacky);

	CASE SC_OvlCentrovacky.Step OF

		0:
			SC_OvlCentrovacky.StepName:= '0 - Nulovanie';
			Centrovacku_VYSUN:= FALSE;
			Centrovacku_ZASUN:= FALSE;
//			P4_FunkcnyTestA.OUT.VysunCentrovanie_YV183:= FALSE;
//			P4_FunkcnyTestA.OUT.ZasunCentrovanie_YV184:= FALSE;

			IF SC_P4_FunkcnyTestA.Step <> 0 THEN
				SC_OvlCentrovacky.ResetStep:= TRUE;
				SC_OvlCentrovacky.Step:= 1;
			END_IF

		1:
			SC_OvlCentrovacky.StepName:= '1 - Rozhodnutie o cinnosti';
			IF Centrovacku_VYSUN THEN
				SC_OvlCentrovacky.Step:= 10;
			ELSIF Centrovacku_ZASUN THEN
				SC_OvlCentrovacky.Step:= 20;
			END_IF

		10:
			SC_OvlCentrovacky.StepName:= '10 - Vysunutie centrovacky';
			SC_OvlCentrovacky.IdleTime.PT:= T#3s;
			SC_OvlCentrovacky.AlarmTime.PT:= T#3s;

			IF P4_FunkcnyTestA.Automat THEN
				SC_OvlCentrovacky.AlarmTime.IN:= TRUE;
			ELSE
				SC_OvlCentrovacky.IdleTime.IN:= TRUE;
			END_IF

			IF NOT SC_OvlCentrovacky.Switch1 THEN
				P4_FunkcnyTestA.OUT.ZasunCentrovanie_YV184:= FALSE;
				P4_FunkcnyTestA.OUT.VysunCentrovanie_YV183:= TRUE;
				SC_OvlCentrovacky.Switch1:= TRUE;
			END_IF

			IF P4_FunkcnyTestA.IN.Centrovanie_VYSUNUTE_MS29 OR SC_OvlCentrovacky.IdleTime.Q THEN
				SC_OvlCentrovacky.ResetStep:= TRUE;
				SC_OvlCentrovacky.Step:= 0;
			ELSIF SC_OvlCentrovacky.AlarmTime.Q THEN
				P34_Alarmy[400]:= TRUE;
				P4_PoruchaST1:= TRUE;
			END_IF

		20:
			SC_OvlCentrovacky.StepName:= '20 - Zasunutie centrovacky';
			SC_OvlCentrovacky.IdleTime.PT:= T#3s;
			SC_OvlCentrovacky.AlarmTime.PT:= T#3s;

			IF P4_FunkcnyTestA.Automat THEN
				SC_OvlCentrovacky.AlarmTime.IN:= TRUE;
			ELSE
				SC_OvlCentrovacky.IdleTime.IN:= TRUE;
			END_IF

			IF NOT SC_OvlCentrovacky.Switch1 THEN
				P4_FunkcnyTestA.OUT.VysunCentrovanie_YV183:= FALSE;
				P4_FunkcnyTestA.OUT.ZasunCentrovanie_YV184:= TRUE;
				SC_OvlCentrovacky.Switch1:= TRUE;
			END_IF

			IF P4_FunkcnyTestA.IN.Centrovanie_ZASUNUTE_MS27 OR SC_OvlCentrovacky.IdleTime.Q THEN
				SC_OvlCentrovacky.ResetStep:= TRUE;
				SC_OvlCentrovacky.Step:= 0;
			ELSIF SC_OvlCentrovacky.AlarmTime.Q THEN
				P34_Alarmy[401]:= TRUE;
				P4_PoruchaST1:= TRUE;
			END_IF

	END_CASE

END_ACTION
```

#### OvlHornychKontaktov.st
```iecst
ACTION OvlHornychKontaktov:

	//Volanie funkcie SequenceControl//
	SequenceControl(SC:= SC_OvlHornychKontaktov);

	CASE SC_OvlHornychKontaktov.Step OF

		0:
			SC_OvlHornychKontaktov.StepName:= '0 - Nulovanie';
			HorneKontakty_VYSUN:= FALSE;
			HorneKontakty_ZASUN:= FALSE;
//			P4_FunkcnyTestA.OUT.HorneKontakty_VYSUN_YV178:= FALSE;
//			P4_FunkcnyTestA.OUT.HorneKontakty_ZASUN_YV177:= FALSE;

			IF SC_P4_FunkcnyTestA.Step <> 0 THEN
				SC_OvlHornychKontaktov.ResetStep:= TRUE;
				SC_OvlHornychKontaktov.Step:= 1;
			END_IF

		1:
			SC_OvlHornychKontaktov.StepName:= '1 - Rozhodnutie o cinnosti';
			IF HorneKontakty_VYSUN THEN
				SC_OvlHornychKontaktov.Step:= 10;
			ELSIF HorneKontakty_ZASUN THEN
				SC_OvlHornychKontaktov.Step:= 20;
			END_IF

		10:
			SC_OvlHornychKontaktov.StepName:= '10 - Vysunutie hornych kontaktov';
			SC_OvlHornychKontaktov.IdleTime.PT:= T#5s;
			SC_OvlHornychKontaktov.AlarmTime.PT:= T#10s;

			IF P4_FunkcnyTestA.Automat THEN
				SC_OvlHornychKontaktov.AlarmTime.IN:= TRUE;
			ELSE
				SC_OvlHornychKontaktov.IdleTime.IN:= TRUE;
			END_IF

			IF NOT SC_OvlHornychKontaktov.Switch1 THEN
				P4_FunkcnyTestA.OUT.HorneKontakty_ZASUN_YV177:= FALSE;
				P4_FunkcnyTestA.OUT.HorneKontakty_VYSUN_YV178:= TRUE;
				SC_OvlHornychKontaktov.Switch1:= TRUE;
			END_IF

			IF P4_FunkcnyTestA.IN.HorneKontakty_VYSUNUTE_MS25 OR SC_OvlHornychKontaktov.IdleTime.Q THEN
				SC_OvlHornychKontaktov.ResetStep:= TRUE;
				SC_OvlHornychKontaktov.Step:= 0;
			ELSIF SC_OvlHornychKontaktov.AlarmTime.Q THEN
				P34_Alarmy[419]:= TRUE;
				P4_PoruchaST1:= TRUE;
			END_IF

		20:
			SC_OvlHornychKontaktov.StepName:= '20 - Zasunutie hornych kontaktov';
			SC_OvlHornychKontaktov.IdleTime.PT:= T#5s;
			SC_OvlHornychKontaktov.AlarmTime.PT:= T#10s;

			IF P4_FunkcnyTestA.Automat THEN
				SC_OvlHornychKontaktov.AlarmTime.IN:= TRUE;
			ELSE
				SC_OvlHornychKontaktov.IdleTime.IN:= TRUE;
			END_IF

			IF NOT SC_OvlHornychKontaktov.Switch1 THEN
				P4_FunkcnyTestA.OUT.HorneKontakty_VYSUN_YV178:= FALSE;
				P4_FunkcnyTestA.OUT.HorneKontakty_ZASUN_YV177:= TRUE;
				SC_OvlHornychKontaktov.Switch1:= TRUE;
			END_IF

			IF P4_FunkcnyTestA.IN.HorneKontakty_ZASUNUTE_MS23 OR SC_OvlHornychKontaktov.IdleTime.Q THEN
				SC_OvlHornychKontaktov.ResetStep:= TRUE;
				SC_OvlHornychKontaktov.Step:= 0;
			ELSIF SC_OvlHornychKontaktov.AlarmTime.Q THEN
				P34_Alarmy[420]:= TRUE;
				P4_PoruchaST1:= TRUE;
			END_IF

	END_CASE

END_ACTION
```

#### OvlSpodnychKontaktov.st
```iecst
ACTION OvlSpodnychKontaktov:

	//Volanie funkcie SequenceControl//
	SequenceControl(SC:= SC_OvlSpodnychKontaktov);

	CASE SC_OvlSpodnychKontaktov.Step OF

		0:
			SC_OvlSpodnychKontaktov.StepName:= '0 - Nulovanie';
			SpodneKontakty_VYSUN:= FALSE;
			SpodneKontakty_ZASUN:= FALSE;
//			P4_FunkcnyTestA.OUT.SpodneKontakty_VYSUN_YV182:= FALSE;
//			P4_FunkcnyTestA.OUT.SpodneKontakty_ZASUN_YV181:= FALSE;

			IF SC_P4_FunkcnyTestA.Step <> 0 THEN
				SC_OvlSpodnychKontaktov.ResetStep:= TRUE;
				SC_OvlSpodnychKontaktov.Step:= 1;
			END_IF

		1:
			SC_OvlSpodnychKontaktov.StepName:= '1 - Rozhodnutie o cinnosti';
			IF SpodneKontakty_VYSUN THEN
				SC_OvlSpodnychKontaktov.Step:= 10;
			ELSIF SpodneKontakty_ZASUN THEN
				SC_OvlSpodnychKontaktov.Step:= 20;
			END_IF

		10:
			SC_OvlSpodnychKontaktov.StepName:= '10 - Vysunutie spodnych kontaktov';
			SC_OvlSpodnychKontaktov.IdleTime.PT:= T#5s;
			SC_OvlSpodnychKontaktov.AlarmTime.PT:= T#10s;

			IF P4_FunkcnyTestA.Automat THEN
				SC_OvlSpodnychKontaktov.AlarmTime.IN:= TRUE;
			ELSE
				SC_OvlSpodnychKontaktov.IdleTime.IN:= TRUE;
			END_IF

			IF NOT SC_OvlSpodnychKontaktov.Switch1 THEN
				P4_FunkcnyTestA.OUT.SpodneKontakty_ZASUN_YV181:= FALSE;
				P4_FunkcnyTestA.OUT.SpodneKontakty_VYSUN_YV182:= TRUE;
				SC_OvlSpodnychKontaktov.Switch1:= TRUE;
			END_IF

			IF P4_FunkcnyTestA.IN.SpodneKontakty_VYSUNUTE_MS33 OR SC_OvlSpodnychKontaktov.IdleTime.Q THEN
				SC_OvlSpodnychKontaktov.ResetStep:= TRUE;
				SC_OvlSpodnychKontaktov.Step:= 0;
			ELSIF SC_OvlSpodnychKontaktov.AlarmTime.Q THEN
				P34_Alarmy[421]:= TRUE;
				P4_PoruchaST1:= TRUE;
			END_IF

		20:
			SC_OvlSpodnychKontaktov.StepName:= '20 - Zasunutie spodnych kontaktov';
			SC_OvlSpodnychKontaktov.IdleTime.PT:= T#5s;
			SC_OvlSpodnychKontaktov.AlarmTime.PT:= T#10s;

			IF P4_FunkcnyTestA.Automat THEN
				SC_OvlSpodnychKontaktov.AlarmTime.IN:= TRUE;
			ELSE
				SC_OvlSpodnychKontaktov.IdleTime.IN:= TRUE;
			END_IF

			IF NOT SC_OvlSpodnychKontaktov.Switch1 THEN
				P4_FunkcnyTestA.OUT.SpodneKontakty_VYSUN_YV182:= FALSE;
				P4_FunkcnyTestA.OUT.SpodneKontakty_ZASUN_YV181:= TRUE;
				SC_OvlSpodnychKontaktov.Switch1:= TRUE;
			END_IF

			IF P4_FunkcnyTestA.IN.SpodneKontakty_ZASUNUTE_MS31 OR SC_OvlSpodnychKontaktov.IdleTime.Q THEN
				SC_OvlSpodnychKontaktov.ResetStep:= TRUE;
				SC_OvlSpodnychKontaktov.Step:= 0;
			ELSIF SC_OvlSpodnychKontaktov.AlarmTime.Q THEN
				P34_Alarmy[422]:= TRUE;
				P4_PoruchaST1:= TRUE;
			END_IF

	END_CASE

END_ACTION
```

#### OvlTestera.st
```iecst
ACTION OvlTestera:

	//Parametre komunikácie//
    memcpy(ADR(SKTcpClientTester_0.Params.IPaddrServ),ADR('192.168.122.252'),SIZEOF('192.168.122.252'));
    (*memcpy(ADR(SKTcpClientTester_0.Params.IPaddrServ),ADR('127.0.0.1'),SIZEOF('127.0.0.1'));*)
    SKTcpClientTester_0.Params.IPportClient := 1032;
    SKTcpClientTester_0.Params.IPportServ := 1030;
    SKTcpClientTester_0.Params.RecvTimeout := 10000;
    strcpy(ADR(SKTcpClientTester_0.Params.Packet.data),ADR(dataStr));
    SKTcpClientTester_0();

    Cas_FunkcnyTestA.PT:= T#1M;
    Cas_FunkcnyTestA();

    //Volanie funkcie SequenceControl//
    SequenceControl(SC:= SC_OvlTesteraFT);

    CASE SC_OvlTesteraFT.Step OF

        0:
            SC_OvlTesteraFT.StepName:= '0 - Nulovanie';
            SKTcpClientTester_0.Enable:= TRUE;
            SKTcpClientTester_0.Cmd.Send:= FALSE;
            FV_Test_UKONCENY:= FALSE;
            FV_Test_PocetDopytovTestera:= 0;
            PocetDopytovNaTester:= 0;
            SC_OvlTesteraFT.ResetStep:= TRUE;
            SC_OvlTesteraFT.Step:= 1;

        1:
            SC_OvlTesteraFT.StepName:= '1 - Cakam na spustenie testera';
            IF FV_Test_START THEN
                P4_FunkcnyTestA.STAV.Vysledok_FV_Testu:= '';
                Cas_FunkcnyTestA.IN:= TRUE;
                NameranyCasFunkcnehoTestuA:= 0;
                SC_OvlTesteraFT.Step:= 10;
            END_IF

        10:
            SC_OvlTesteraFT.StepName:= '10 - Dopyt na stav testera - typ 0';
            SC_OvlTesteraFT.IdleTime.PT:= T#300ms;
            SC_OvlTesteraFT.AlarmTime.PT:= T#5s;
            SC_OvlTesteraFT.IdleTime.IN:= TRUE;
            SC_OvlTesteraFT.AlarmTime.IN:= TRUE;

            SKTcpClientTester_0.Params.Packet.type:= 0;
            SKTcpClientTester_0.Params.Packet.workplace:= 49;
            SKTcpClientTester_0.Params.Packet.id:= 1;
            SKTcpClientTester_0.Cmd.Send:= TRUE;

            IF SKTcpClientTester_0.Cmd.Send AND NOT SKTcpClientTester_0.Status.staReceived AND NOT SKTcpClientTester_0.Status.staError THEN
                SC_OvlTesteraFT.ResetStep:= TRUE;
                SC_OvlTesteraFT.Step:= 13;
            ELSIF SC_OvlTesteraFT.AlarmTime.Q AND (SKTcpClientTester_0.Status.staReceived OR SKTcpClientTester_0.Status.staError) THEN
                PocetDopytovNaTester:= PocetDopytovNaTester + 1;
                SC_OvlTesteraFT.ResetStep:= TRUE;
                SC_OvlTesteraFT.Step:= 12;
            END_IF

        12:
            SC_OvlTesteraFT.StepName:= '12 - Dopyt na stav testera - cakam na opatovny dopyt na tester';
            SC_OvlTesteraFT.IdleTime.PT:= T#300ms;
            SC_OvlTesteraFT.AlarmTime.PT:= T#5s;
            SC_OvlTesteraFT.IdleTime.IN:= TRUE;
            SKTcpClientTester_0.Cmd.Send:= FALSE;

            IF PocetDopytovNaTester < 10 THEN
                IF SC_OvlTesteraFT.IdleTime.Q THEN
                    SC_OvlTesteraFT.ResetStep:= TRUE;
                    SC_OvlTesteraFT.Step:= 10;
                END_IF
            ELSE
                P4_FunkcnyTestA.STAV.Vysledok_FV_Testu:= 'NG';
                FV_Test_UKONCENY:= TRUE;
                SC_OvlTesteraFT.ResetStep:= TRUE;
                SC_OvlTesteraFT.Step:= 100;
            END_IF

        13:
            SC_OvlTesteraFT.StepName:= '13 - Odpoved na stav testera - typ 0';
            SC_OvlTesteraFT.IdleTime.PT:= T#300ms;
            SC_OvlTesteraFT.AlarmTime.PT:= T#10s;
            SC_OvlTesteraFT.IdleTime.IN:= TRUE;

            IF SKTcpClientTester_0.Status.staReceived AND SKTcpClientTester_0.Status.DataRecv[2]= 0 AND SKTcpClientTester_0.Status.DataRecv[5]= 2 THEN
                SKTcpClientTester_0.Cmd.Send:= FALSE;
                SC_OvlTesteraFT.ResetStep:= TRUE;
                SC_OvlTesteraFT.Step:= 15;
            ELSIF SKTcpClientTester_0.Status.staReceived AND SKTcpClientTester_0.Status.DataRecv[2]= 0 AND SKTcpClientTester_0.Status.DataRecv[5]= 1 THEN
                SKTcpClientTester_0.Cmd.Send:= FALSE;
                IF SC_OvlTesteraFT.IdleTime.Q THEN
                    SC_OvlTesteraFT.ResetStep:= TRUE;
                    SC_OvlTesteraFT.Step:= 10;
                END_IF
            ELSIF SKTcpClientTester_0.Status.staReceived AND SKTcpClientTester_0.Status.DataRecv[2]= 0 AND SKTcpClientTester_0.Status.DataRecv[5]= 0 THEN
                SKTcpClientTester_0.Cmd.Send:= FALSE;
                IF SC_OvlTesteraFT.IdleTime.Q THEN
                    SC_OvlTesteraFT.ResetStep:= TRUE;
                    SC_OvlTesteraFT.Step:= 10;
                END_IF
            ELSIF SKTcpClientTester_0.Status.staError THEN
                SKTcpClientTester_0.Cmd.Send:= FALSE;
                P4_FunkcnyTestA.STAV.Vysledok_FV_Testu:= 'NG';
                FV_Test_UKONCENY:= TRUE;
                SC_OvlTesteraFT.ResetStep:= TRUE;
                SC_OvlTesteraFT.Step:= 100;
            END_IF

        15:
            SC_OvlTesteraFT.StepName:= '15 - Poslanie QR kodu Power CP - typ 1';
            SC_OvlTesteraFT.IdleTime.PT:= T#300ms;
            SC_OvlTesteraFT.AlarmTime.PT:= T#10s;
            SC_OvlTesteraFT.IdleTime.IN:= TRUE;

            SKTcpClientTester_0.Params.Packet.type:= 1;
            SKTcpClientTester_0.Params.Packet.workplace:= 49;
            SKTcpClientTester_0.Params.Packet.id:= 1;
            dataStr:= Paletka[i].PAR.QRkodPowerCP;
            SKTcpClientTester_0.Cmd.Send:= TRUE;

            IF SKTcpClientTester_0.Cmd.Send AND NOT SKTcpClientTester_0.Status.staReceived AND NOT SKTcpClientTester_0.Status.staError THEN
                SC_OvlTesteraFT.ResetStep:= TRUE;
                SC_OvlTesteraFT.Step:= 18;
            END_IF

        18:
            SC_OvlTesteraFT.StepName:= '18 - Odpoved na poslanie QR kodu - typ 1';
            SC_OvlTesteraFT.IdleTime.PT:= T#300ms;
            SC_OvlTesteraFT.AlarmTime.PT:= T#10s;
            SC_OvlTesteraFT.IdleTime.IN:= TRUE;

            IF SKTcpClientTester_0.Status.staReceived AND SKTcpClientTester_0.Status.DataRecv[2]= 1 AND SKTcpClientTester_0.Status.DataRecv[5]= 0 THEN
                SKTcpClientTester_0.Cmd.Send:= FALSE;
                SC_OvlTesteraFT.ResetStep:= TRUE;
                SC_OvlTesteraFT.Step:= 20;
            ELSIF SKTcpClientTester_0.Status.staReceived AND SKTcpClientTester_0.Status.DataRecv[2]= 1 AND SKTcpClientTester_0.Status.DataRecv[5]= 2 THEN
                SKTcpClientTester_0.Cmd.Send:= FALSE;
                IF SC_OvlTesteraFT.IdleTime.Q THEN
                    SC_OvlTesteraFT.ResetStep:= TRUE;
                    SC_OvlTesteraFT.Step:= 15;
                END_IF
            ELSIF SKTcpClientTester_0.Status.staReceived AND SKTcpClientTester_0.Status.DataRecv[2]= 1 AND SKTcpClientTester_0.Status.DataRecv[5]= 1 THEN
                SKTcpClientTester_0.Cmd.Send:= FALSE;
                P4_FunkcnyTestA.STAV.Vysledok_FV_Testu:= 'NG';
                FV_Test_UKONCENY:= TRUE;
                SC_OvlTesteraFT.ResetStep:= TRUE;
                SC_OvlTesteraFT.Step:= 100;
            ELSIF SKTcpClientTester_0.Status.staError THEN
                SKTcpClientTester_0.Cmd.Send:= FALSE;
                P4_FunkcnyTestA.STAV.Vysledok_FV_Testu:= 'NG';
                FV_Test_UKONCENY:= TRUE;
                SC_OvlTesteraFT.ResetStep:= TRUE;
                SC_OvlTesteraFT.Step:= 100;
            END_IF

        20:
            SC_OvlTesteraFT.StepName:= '20 - Dopyt na stav testera - typ 0';
            SC_OvlTesteraFT.IdleTime.PT:= T#300ms;
            SC_OvlTesteraFT.AlarmTime.PT:= T#10s;
            SC_OvlTesteraFT.IdleTime.IN:= TRUE;

            SKTcpClientTester_0.Params.Packet.type:= 0;
            SKTcpClientTester_0.Params.Packet.workplace:= 49;
            SKTcpClientTester_0.Params.Packet.id:= 1;
            SKTcpClientTester_0.Cmd.Send:= TRUE;

            IF SKTcpClientTester_0.Cmd.Send AND NOT SKTcpClientTester_0.Status.staReceived AND NOT SKTcpClientTester_0.Status.staError THEN
                SC_OvlTesteraFT.ResetStep:= TRUE;
                SC_OvlTesteraFT.Step:= 23;
            END_IF

        23:
            SC_OvlTesteraFT.StepName:= '23 - Odpoved na stav testera - typ 0';
            SC_OvlTesteraFT.IdleTime.PT:= T#300ms;
            SC_OvlTesteraFT.AlarmTime.PT:= T#10s;
            SC_OvlTesteraFT.IdleTime.IN:= TRUE;

            IF SKTcpClientTester_0.Status.staReceived AND SKTcpClientTester_0.Status.DataRecv[2]= 0 AND SKTcpClientTester_0.Status.DataRecv[5]= 3 THEN
                SKTcpClientTester_0.Cmd.Send:= FALSE;
                IF SC_OvlTesteraFT.IdleTime.Q THEN
                    SC_OvlTesteraFT.ResetStep:= TRUE;
                    SC_OvlTesteraFT.Step:= 20;
                END_IF
            ELSIF SKTcpClientTester_0.Status.staReceived AND SKTcpClientTester_0.Status.DataRecv[2]= 0 AND SKTcpClientTester_0.Status.DataRecv[5]= 4 THEN
                SKTcpClientTester_0.Cmd.Send:= FALSE;
                SC_OvlTesteraFT.ResetStep:= TRUE;
                SC_OvlTesteraFT.Step:= 25;
            ELSIF SKTcpClientTester_0.Status.staReceived AND SKTcpClientTester_0.Status.DataRecv[2]= 0 AND SKTcpClientTester_0.Status.DataRecv[5]= 0 THEN
                SKTcpClientTester_0.Cmd.Send:= FALSE;
                P4_FunkcnyTestA.STAV.Vysledok_FV_Testu:= 'NG';
                FV_Test_UKONCENY:= TRUE;
                SC_OvlTesteraFT.ResetStep:= TRUE;
                SC_OvlTesteraFT.Step:= 100;
            ELSIF SKTcpClientTester_0.Status.staError THEN
                SKTcpClientTester_0.Cmd.Send:= FALSE;
                P4_FunkcnyTestA.STAV.Vysledok_FV_Testu:= 'NG';
                FV_Test_UKONCENY:= TRUE;
                SC_OvlTesteraFT.ResetStep:= TRUE;
                SC_OvlTesteraFT.Step:= 100;
            END_IF

        25:
            SC_OvlTesteraFT.StepName:= '25 - Dopyt na vysledok testu - typ 2';
            SC_OvlTesteraFT.IdleTime.PT:= T#300ms;
            SC_OvlTesteraFT.AlarmTime.PT:= T#10s;
            SC_OvlTesteraFT.IdleTime.IN:= TRUE;

            SKTcpClientTester_0.Params.Packet.type:= 2;
            SKTcpClientTester_0.Params.Packet.workplace:= 49;
            SKTcpClientTester_0.Params.Packet.id:= 1;
            SKTcpClientTester_0.Cmd.Send:= TRUE;

            IF SKTcpClientTester_0.Cmd.Send AND NOT SKTcpClientTester_0.Status.staReceived AND NOT SKTcpClientTester_0.Status.staError THEN
                SC_OvlTesteraFT.ResetStep:= TRUE;
                SC_OvlTesteraFT.Step:= 28;
            END_IF

        28:
            SC_OvlTesteraFT.StepName:= '28 - Odpoved na vysledok testu - typ 2';
            SC_OvlTesteraFT.IdleTime.PT:= T#300ms;
            SC_OvlTesteraFT.AlarmTime.PT:= T#10s;
            SC_OvlTesteraFT.IdleTime.IN:= TRUE;

            IF SKTcpClientTester_0.Status.staReceived AND SKTcpClientTester_0.Status.DataRecv[2]= 2 AND SKTcpClientTester_0.Status.DataRecv[5]= 1 THEN
                SKTcpClientTester_0.Cmd.Send:= FALSE;
                P4_FunkcnyTestA.STAV.Vysledok_FV_Testu:= 'OK';
                SC_OvlTesteraFT.ResetStep:= TRUE;
                SC_OvlTesteraFT.Step:= 30;
            ELSIF SKTcpClientTester_0.Status.staReceived AND SKTcpClientTester_0.Status.DataRecv[2]= 2 AND SKTcpClientTester_0.Status.DataRecv[5]= 2 THEN
                SKTcpClientTester_0.Cmd.Send:= FALSE;
                P4_FunkcnyTestA.STAV.Vysledok_FV_Testu:= 'NG';
                SC_OvlTesteraFT.ResetStep:= TRUE;
                SC_OvlTesteraFT.Step:= 30;
            ELSIF SKTcpClientTester_0.Status.staReceived AND SKTcpClientTester_0.Status.DataRecv[2]= 2 AND SKTcpClientTester_0.Status.DataRecv[5]= 0 THEN
                SKTcpClientTester_0.Cmd.Send:= FALSE;
                IF SC_OvlTesteraFT.IdleTime.Q THEN
                    SC_OvlTesteraFT.ResetStep:= TRUE;
                    SC_OvlTesteraFT.Step:= 25;
                END_IF
            ELSIF SKTcpClientTester_0.Status.staReceived AND SKTcpClientTester_0.Status.DataRecv[2]= 2 AND SKTcpClientTester_0.Status.DataRecv[5]= 3 THEN
                SKTcpClientTester_0.Cmd.Send:= FALSE;
                IF SC_OvlTesteraFT.IdleTime.Q THEN
                    SC_OvlTesteraFT.ResetStep:= TRUE;
                    SC_OvlTesteraFT.Step:= 25;
                END_IF
            ELSIF SKTcpClientTester_0.Status.staError THEN
                SKTcpClientTester_0.Cmd.Send:= FALSE;
                P4_FunkcnyTestA.STAV.Vysledok_FV_Testu:= 'NG';
                FV_Test_UKONCENY:= TRUE;
                SC_OvlTesteraFT.ResetStep:= TRUE;
                SC_OvlTesteraFT.Step:= 100;
            END_IF

        30:
            SC_OvlTesteraFT.StepName:= '30 - Potvrdenie precitanie vysledkov testu - typ 3';
            SC_OvlTesteraFT.IdleTime.PT:= T#300ms;
            SC_OvlTesteraFT.AlarmTime.PT:= T#10s;
            SC_OvlTesteraFT.IdleTime.IN:= TRUE;

            SKTcpClientTester_0.Params.Packet.type:= 3;
            SKTcpClientTester_0.Params.Packet.workplace:= 49;
            SKTcpClientTester_0.Params.Packet.id:= 1;
            SKTcpClientTester_0.Cmd.Send:= TRUE;

            IF SKTcpClientTester_0.Cmd.Send AND NOT SKTcpClientTester_0.Status.staReceived AND NOT SKTcpClientTester_0.Status.staError THEN
                SC_OvlTesteraFT.ResetStep:= TRUE;
                SC_OvlTesteraFT.Step:= 33;
            END_IF

        33:
            SC_OvlTesteraFT.StepName:= '33 - Odpoved testera na potvrdenie vysledkov - typ 3';
            SC_OvlTesteraFT.IdleTime.PT:= T#500ms;
            SC_OvlTesteraFT.AlarmTime.PT:= T#10s;

            IF SKTcpClientTester_0.Status.staReceived AND SKTcpClientTester_0.Status.DataRecv[2]= 3 AND SKTcpClientTester_0.Status.DataRecv[5]= 0 THEN
                SKTcpClientTester_0.Cmd.Send:= FALSE;
                FV_Test_UKONCENY:= TRUE;
                SC_OvlTesteraFT.ResetStep:= TRUE;
                SC_OvlTesteraFT.Step:= 100;
            ELSIF SKTcpClientTester_0.Status.staReceived AND SKTcpClientTester_0.Status.DataRecv[2]= 3 AND SKTcpClientTester_0.Status.DataRecv[5]= 1 THEN
                P4_FunkcnyTestA.STAV.Vysledok_FV_Testu:= 'NG';
                FV_Test_UKONCENY:= TRUE;
                SKTcpClientTester_0.Cmd.Send:= FALSE;
                SC_OvlTesteraFT.ResetStep:= TRUE;
                SC_OvlTesteraFT.Step:= 100;
            ELSIF SKTcpClientTester_0.Status.staError THEN
                SKTcpClientTester_0.Cmd.Send:= FALSE;
                SC_OvlTesteraFT.ResetStep:= TRUE;
                SC_OvlTesteraFT.Step:= 100;
            END_IF

        100:
            SC_OvlTesteraFT.StepName:= '100 - Cakam na zrusenie signalu start testovania';
            SC_OvlTesteraFT.IdleTime.PT:= T#3s;
            SC_OvlTesteraFT.AlarmTime.PT:= T#10s;

            NameranyCasFunkcnehoTestuA:= Cas_FunkcnyTestA.ET;
            Cas_FunkcnyTestA.IN:= FALSE;

            IF NOT FV_Test_START THEN
                SC_OvlTesteraFT.ResetStep:= TRUE;
                SC_OvlTesteraFT.Step:= 0;
            END_IF

    END_CASE

END_ACTION
```

### Program Logical/Program/Pracovisko_4/P4_StoperFunkcnyTestB (IEC)

#### Main.st - Init, cyclic, exit code
```iecst
PROGRAM _INIT
    Triger_0:= FALSE;
    Triger_1:= FALSE;

    P4_FunkcnyTestB.STAV.Tester_ON:= TRUE;
    P4_FunkcnyTestB.OUT.HorneKontakty_ZASUN_YV185:= TRUE;
END_PROGRAM

PROGRAM _CYCLIC

	//Volanie podprogramov//
    OvlCentrovacky;
    IOLinkKomunikacia;
    OvlHornychKontaktov;
    OvlSpodnychKontaktov;
    OvlTestera;

    //Volanie funkcie SequenceControl//
    SequenceControl(SC:= SC_P4_FunkcnyTestB);

    //Príznak funkčný test A východzia pozícia//
    IF P4_FunkcnyTestB.IN.Centrovanie_ZASUNUTE_MS28 AND P4_FunkcnyTestB.IN.HorneKontakty_ZASUNUTE_MS24 AND P4_FunkcnyTestB.IN.SpodneKontakty_ZASUNUTE_MS32 THEN
        P4_FunkcnyTestB_VychodziaPozicia:= TRUE;
    ELSE
        P4_FunkcnyTestB_VychodziaPozicia:= FALSE;
    END_IF

    //Reset sekcie //
    IF NOT Safety.STAV.P4_ZonaBunky_AKTIVNA THEN
        SC_P4_FunkcnyTestB.Step:= 0;
    ELSIF P4_FunkcnyTestB.Reset THEN
        SC_P4_FunkcnyTestB.Step:= 0;
        P4_FunkcnyTestB.Reset:= FALSE;
    END_IF

    //Porucha stanice//
    IF P4_PoruchaST2 AND NOT Triger_0 THEN
        Triger_0:= TRUE;
        SC_P4_FunkcnyTestB.Step:= 0;
     END_IF

    IF NOT P4_PoruchaST2 THEN
        Triger_0:= FALSE;
    END_IF

    //Čas testovania//
    CasTestovania.PT:= T#5M;
    CasTestovania();
    NameranyCasTestovania;

    CASE SC_P4_FunkcnyTestB.Step OF

        0:
            SC_P4_FunkcnyTestB.StepName:='0 - Nulovanie';
            SC_OvlCentrovacky.Step:= 0;
            SC_OvlHornychKontaktov.Step:= 0;
            SC_OvlSpodnychKontaktov.Step:= 0;
            P4_FunkcnyTestB.Automat:= FALSE;
            P4_FunkcnyTestB.KoniecCyklu:= FALSE;
            P4_FunkcnyTestB.Manual:= FALSE;
            P4_FunkcnyTestB.STAV.PoINIT:= FALSE;
            P4_FunkcnyTestB.OUT.KontaktyTestera_VYSUN_YV172:= FALSE;
            P4_FunkcnyTestB.OUT.OdpruzenieKontaktov_VYPNI_YV188:= TRUE;
            P4_FunkcnyTestB.OUT.OdpruzenieKontaktov_ZAPNI_YV187:= FALSE;
            P4_FunkcnyTestB.OUT.ZasunStoper_YV164:= FALSE;
            PrecitaneCisloPaletky:= '';
            FV_Test_START:= FALSE;
            FV_Test_UKONCENY:= FALSE;
            Taktime_FunkcnyTestB.CMD.START_Merania_1:= FALSE;
            Taktime_FunkcnyTestB.CMD.START_Merania_2:= FALSE;
			P4_FunkcnyTestB.STAV.PrebiehaVyvezeniePaletky:= FALSE;
			P4_FunkcnyTestB_ZATVOR:= FALSE;
			P4_FunkcnyTestB_OTVOR:= FALSE;
            TestovaciKus:= FALSE;
            Revork:= FALSE;
            P4_FunkcnyTestB.OUT.KOM_StanicaA_StartTestovania:= FALSE;
            CasTestovania.IN:= FALSE;
            P4_FunkcnyTestB.RR_TestovanieFunkcnehoTestu:= FALSE;
            P4_FunkcnyTestB.RR_VysunKontaktyTestera:= FALSE;
            P4_FunkcnyTestB.RR_ZapniOdpruzenieKontaktov:= FALSE;
            P4_FunkcnyTestB.RR_OtvorTester:= FALSE;
            P4_FunkcnyTestB.RR_ZatvorTester:= FALSE;
            PocetOpakovaniTestu:= 0;
            OpakovanyTest:= FALSE;

            IF Safety.STAV.P4_ZonaBunky_AKTIVNA AND NOT P4_Pracovisko.STAV.PORUCHA AND P4_Pracovisko.IN.PrivodVzduchu_SnimacTlaku_S15 THEN
                SC_P4_FunkcnyTestB.ResetStep:= TRUE;
                SC_P4_FunkcnyTestB.Step:= 1;
            END_IF

        1:
            SC_P4_FunkcnyTestB.StepName:='1 - Cakam na spustenie vyroby';
            P4_FunkcnyTestB.KoniecCyklu:= FALSE;
            IF P4_FunkcnyTestB.Automat THEN
                SC_P4_FunkcnyTestB.Step:= 2;
            ELSIF P4_FunkcnyTestB.Manual THEN
				SC_P4_FunkcnyTestB.Step:= 700;
			ELSIF P4_FunkcnyTestB_ZATVOR THEN
				SC_P4_FunkcnyTestB.Step:= 720;
			ELSIF P4_FunkcnyTestB_OTVOR THEN
				SC_P4_FunkcnyTestB.Step:= 750;
            END_IF

            //********************************************************Inicializácia****************************************************************************//

        2:
            SC_P4_FunkcnyTestB.StepName:='2 - Inicializacia - cakam na spustenie inicializacie';
            SC_P4_FunkcnyTestB.IdleTime.PT:= T#2s;
            SC_P4_FunkcnyTestB.AlarmTime.PT:= T#5s;

            SC_P4_FunkcnyTestB.IdleTime.IN:= TRUE;

            IF SC_P4_FunkcnyTestB.IdleTime.Q THEN
                SC_P4_FunkcnyTestB.ResetStep:= TRUE;
                SC_P4_FunkcnyTestB.Step:= 3;
            END_IF

        3:
            SC_P4_FunkcnyTestB.StepName:='3 - Inicializacia - zasunutie hornych kontaktov';
            SC_P4_FunkcnyTestB.IdleTime.PT:= T#2s;
            SC_P4_FunkcnyTestB.AlarmTime.PT:= T#5s;

            IF NOT SC_P4_FunkcnyTestB.Switch1 THEN
                HorneKontakty_ZASUN:= TRUE;
                SC_P4_FunkcnyTestB.Switch1:= TRUE;
            END_IF

            IF P4_FunkcnyTestB.IN.HorneKontakty_ZASUNUTE_MS24 THEN
                SC_P4_FunkcnyTestB.ResetStep:= TRUE;
                SC_P4_FunkcnyTestB.Step:= 5;
            END_IF

        5:
            SC_P4_FunkcnyTestB.StepName:='5 - Inicializacia - zasunutie spodnych kontaktov';
            SC_P4_FunkcnyTestB.IdleTime.PT:= T#2s;
            SC_P4_FunkcnyTestB.AlarmTime.PT:= T#5s;

            IF NOT SC_P4_FunkcnyTestB.Switch1 THEN
                SpodneKontakty_ZASUN:= TRUE;
                SC_P4_FunkcnyTestB.Switch1:= TRUE;
            END_IF

            IF P4_FunkcnyTestB.IN.SpodneKontakty_ZASUNUTE_MS32 THEN
                SC_P4_FunkcnyTestB.ResetStep:= TRUE;
                SC_P4_FunkcnyTestB.Step:= 8;
            END_IF

        8:
            SC_P4_FunkcnyTestB.StepName:='8 - Inicializacia - zasunutie centrovacky';
            SC_P4_FunkcnyTestB.IdleTime.PT:= T#4s;
            SC_P4_FunkcnyTestB.AlarmTime.PT:= T#5s;

            IF NOT SC_P4_FunkcnyTestB.Switch1 THEN
                Centrovacku_ZASUN:= TRUE;
                SC_P4_FunkcnyTestB.Switch1:= TRUE;
            END_IF

            IF P4_FunkcnyTestB.IN.Centrovanie_ZASUNUTE_MS28 AND P4_Dopravniky.STAV.PoINIT THEN
                SC_P4_FunkcnyTestB.ResetStep:= TRUE;
                SC_P4_FunkcnyTestB.Step:= 10;
            END_IF

        10:
            SC_P4_FunkcnyTestB.StepName:='10 - Inicializacia - kontrola kontaktov funkcneho testu';
            SC_P4_FunkcnyTestB.IdleTime.PT:= T#4s;
            SC_P4_FunkcnyTestB.AlarmTime.PT:= T#5s;

            IF Linka.PAR.ZvolenyModel = '4F' AND P4_FunkcnyTestB.IN.TypSpodnychKontaktov_4F THEN
                SC_P4_FunkcnyTestB.ResetStep:= TRUE;
                SC_P4_FunkcnyTestB.Step:= 13;
            ELSIF Linka.PAR.ZvolenyModel = '5F' AND P4_FunkcnyTestB.IN.TypSpodnychKontaktov_5F_5H THEN
                SC_P4_FunkcnyTestB.ResetStep:= TRUE;
                SC_P4_FunkcnyTestB.Step:= 13;
            ELSIF Linka.PAR.ZvolenyModel = '5H'AND P4_FunkcnyTestB.IN.TypSpodnychKontaktov_5F_5H THEN
                SC_P4_FunkcnyTestB.ResetStep:= TRUE;
                SC_P4_FunkcnyTestB.Step:= 13;
            ELSE
                P34_Alarmy[438]:= TRUE;
                P4_PoruchaST2:= TRUE;
            END_IF

        13:
            SC_P4_FunkcnyTestB.StepName:='13 - Inicializacia - hladanie paletky';
            SC_P4_FunkcnyTestB.IdleTime.PT:= T#5s;
            SC_P4_FunkcnyTestB.AlarmTime.PT:= T#5s;
            SC_P4_FunkcnyTestB.IdleTime.IN:= TRUE;

            IF P4_FunkcnyTestB.IN.PritomnostPaletky_S11 THEN
                P4_FunkcnyTestA.STAV.PrebiehaVyvezeniePaletky:= FALSE;
                P4_FunkcnyTestB.STAV.PoINIT:= TRUE;
                SC_P4_FunkcnyTestB.ResetStep:= TRUE;
                SC_P4_FunkcnyTestB.Step:= 20;
            ELSIF SC_P4_FunkcnyTestB.IdleTime.Q THEN
                P4_FunkcnyTestB.STAV.PoINIT:= TRUE;
                SC_P4_FunkcnyTestB.ResetStep:= TRUE;
                SC_P4_FunkcnyTestB.Step:= 100;
            END_IF

        20:
            SC_P4_FunkcnyTestB.StepName:='20 - Inicializacia - precitanie cisla paletky';
            SC_P4_FunkcnyTestB.IdleTime.PT:= T#200ms;
            SC_P4_FunkcnyTestB.AlarmTime.PT:= T#5s;
            SC_P4_FunkcnyTestB.IdleTime.IN:= TRUE;

            IF SC_P4_FunkcnyTestB.IdleTime.Q THEN
                PrecitaneCisloPaletky:= USINT_TO_STRING(P4_FunkcnyTestB.IN.PrecitaneCisloPaletky_S11);
                i:= 0;
                SC_P4_FunkcnyTestB.ResetStep:= TRUE;
                SC_P4_FunkcnyTestB.Step:= 23;
            END_IF

        23:
            SC_P4_FunkcnyTestB.StepName:='23 - Inicializacia - priradenie indexu paletky na zaklade precitanej hodnoty';
            SC_P4_FunkcnyTestB.IdleTime.PT:= T#200ms;
            SC_P4_FunkcnyTestB.AlarmTime.PT:= T#5s;

            IF PrecitaneCisloPaletky = '171' THEN
                i:= 1;
            ELSIF PrecitaneCisloPaletky = '164' THEN
                i:= 2;
            ELSIF PrecitaneCisloPaletky = '181' THEN
                i:= 3;
            ELSIF PrecitaneCisloPaletky = '168' THEN
                i:= 4;
            ELSIF PrecitaneCisloPaletky = '140' THEN
                i:= 5;
            ELSIF PrecitaneCisloPaletky = '110' THEN
                i:= 6;
            ELSIF PrecitaneCisloPaletky = '156' THEN
                i:= 7;
            ELSIF PrecitaneCisloPaletky = '127' THEN
                i:= 8;
            ELSIF PrecitaneCisloPaletky = '139' THEN
                i:= 9;
            ELSIF PrecitaneCisloPaletky = '131' THEN
                i:= 10;
            ELSIF PrecitaneCisloPaletky = '178' THEN
                i:= 11;
            ELSIF PrecitaneCisloPaletky = '206' THEN
                i:= 12;
            ELSIF PrecitaneCisloPaletky = '119' THEN
                i:= 13;
            ELSIF PrecitaneCisloPaletky = '163' THEN
                i:= 14;
            ELSIF PrecitaneCisloPaletky = '128' THEN
                i:= 15;
            ELSIF PrecitaneCisloPaletky = '175' THEN
                i:= 16;
            ELSIF PrecitaneCisloPaletky = '138' THEN
                i:= 17;
            ELSE
                P34_Alarmy[429]:= TRUE;
                P4_PoruchaST2:= TRUE;
            END_IF

            IF i<> 0 THEN
                Paletka[i].PAR.CisloPaletky:= USINT_TO_STRING(i);
                PrecitaneCisloPaletky:= '';
                SC_P4_FunkcnyTestB.ResetStep:= TRUE;
                SC_P4_FunkcnyTestB.Step:= 30;
            END_IF

        30:
            SC_P4_FunkcnyTestB.StepName:='30 - Inicializacia - kontrola stavu paletky';
            SC_P4_FunkcnyTestB.IdleTime.PT:= T#200ms;
            SC_P4_FunkcnyTestB.AlarmTime.PT:= T#5s;

            IF Paletka[i].PAR.TestovaciKus AND Paletka[i].PAR.CisloTestovacejStanice = 'ST_FT1,FT2' THEN
                IF P4_FunkcnyTestB.STAV.Tester_ON THEN
                    TestovaciKus:= TRUE;
                    P4_FunkcnyTestB.STAV.PoINIT:= TRUE;
                    SC_P4_FunkcnyTestB.ResetStep:= TRUE;
                    SC_P4_FunkcnyTestB.Step:= 118;
                ELSE
                    P4_FunkcnyTestB.STAV.PoINIT:= TRUE;
                    SC_P4_FunkcnyTestB.ResetStep:= TRUE;
                    SC_P4_FunkcnyTestB.Step:= 560;
                END_IF
            ELSIF Paletka[i].PAR.TestovaciKus AND Paletka[i].PAR.CisloTestovacejStanice <> 'ST_FT1,FT2' THEN
                P4_FunkcnyTestB.STAV.PoINIT:= TRUE;
                SC_P4_FunkcnyTestB.ResetStep:= TRUE;
                SC_P4_FunkcnyTestB.Step:= 560;
            ELSIF Paletka[i].PAR.RevorkovyKus AND Paletka[i].PAR.CisloRevorkovejStanice = 'ST_FT1,FT2' THEN
                IF P4_FunkcnyTestB.STAV.Tester_ON THEN
                    Revork:= TRUE;
                    P4_FunkcnyTestB.STAV.PoINIT:= TRUE;
                    SC_P4_FunkcnyTestB.ResetStep:= TRUE;
                    SC_P4_FunkcnyTestB.Step:= 105;
                ELSE
                    P4_FunkcnyTestB.STAV.PoINIT:= TRUE;
                    SC_P4_FunkcnyTestB.ResetStep:= TRUE;
                    SC_P4_FunkcnyTestB.Step:= 560;
                END_IF
            ELSIF Paletka[i].PAR.RevorkovyKus AND Paletka[i].PAR.CisloRevorkovejStanice <> 'ST_FT1,FT2' THEN
                Revork:= FALSE;
                P4_FunkcnyTestB.STAV.PoINIT:= TRUE;
                SC_P4_FunkcnyTestB.ResetStep:= TRUE;
                SC_P4_FunkcnyTestB.Step:= 560;
            ELSIF Paletka[i].PAR.StavPaletky = 'OK' THEN
                SC_P4_FunkcnyTestB.ResetStep:= TRUE;
                SC_P4_FunkcnyTestB.Step:= 33;
            ELSIF Paletka[i].PAR.StavPaletky = 'NG' THEN
                P4_FunkcnyTestB.STAV.PoINIT:= TRUE;
                SC_P4_FunkcnyTestB.ResetStep:= TRUE;
                SC_P4_FunkcnyTestB.Step:= 560;
            END_IF

        33:
            SC_P4_FunkcnyTestB.StepName:='33 - Inicializacia - kontrola ukoncenia testu';
            SC_P4_FunkcnyTestB.IdleTime.PT:= T#200ms;
            SC_P4_FunkcnyTestB.AlarmTime.PT:= T#5s;

            IF Paletka[i].VnutornyStav.FunkcnyTest_Ukonceny THEN
                P4_FunkcnyTestB.STAV.PoINIT:= TRUE;
                SC_P4_FunkcnyTestB.ResetStep:= TRUE;
                SC_P4_FunkcnyTestB.Step:= 560;
            ELSE
                P4_FunkcnyTestB.STAV.PoINIT:= TRUE;
                SC_P4_FunkcnyTestB.ResetStep:= TRUE;
                SC_P4_FunkcnyTestB.Step:= 100;
            END_IF

            //********************************************************Automatický režim****************************************************************************//

        100:
            SC_P4_FunkcnyTestB.StepName:='100 - Automaticky Rezim - cakam na príchod paletky na stoper';
            SC_P4_FunkcnyTestB.IdleTime.PT:= T#200ms;
            SC_P4_FunkcnyTestB.AlarmTime.PT:= T#5s;

            IF P4_FunkcnyTestB.IN.PritomnostPaletky_S11 THEN
                P4_FunkcnyTestA.STAV.PrebiehaVyvezeniePaletky:= FALSE;
            END_IF

            SC_P4_FunkcnyTestB.IdleTime.IN:= P4_FunkcnyTestB.IN.PritomnostPaletky_S11;

            IF EDGEPOS(P4_FunkcnyTestB.IN.PritomnostPaletky_S11)THEN
                IF NOT Taktime_FunkcnyTestB.CMD.START_Merania_1 THEN
                    Taktime_FunkcnyTestB.CMD.START_Merania_1:= TRUE;
                ELSE
                    Taktime_FunkcnyTestB.CMD.ZAPIS_Hodnot_1:= TRUE;
                END_IF
            END_IF

            IF P4_FunkcnyTestB.KoniecCyklu THEN
                SC_P4_FunkcnyTestB.ResetStep:= TRUE;
                SC_P4_FunkcnyTestB.Step:= 0;
            ELSIF SC_P4_FunkcnyTestB.IdleTime.Q THEN
                SC_P4_FunkcnyTestB.ResetStep:= TRUE;
                SC_P4_FunkcnyTestB.Step:= 101;
            END_IF

        101:
            SC_P4_FunkcnyTestB.StepName:='101 - Automaticky Rezim - precitanie cisla paletky';
            SC_P4_FunkcnyTestB.IdleTime.PT:= T#500ms;
            SC_P4_FunkcnyTestB.AlarmTime.PT:= T#5s;
            SC_P4_FunkcnyTestB.IdleTime.IN:= TRUE;

            PrecitaneCisloPaletky:= USINT_TO_STRING(P4_FunkcnyTestB.IN.PrecitaneCisloPaletky_S11);
            i:= 0;
            SC_P4_FunkcnyTestB.ResetStep:= TRUE;
            SC_P4_FunkcnyTestB.Step:= 102;

        102:
            SC_P4_FunkcnyTestB.StepName:='102 - Automaticky Rezim - priradenie indexu paletky na zaklade precitanej hodnoty';
            SC_P4_FunkcnyTestB.IdleTime.PT:= T#200ms;
            SC_P4_FunkcnyTestB.AlarmTime.PT:= T#5s;

            IF PrecitaneCisloPaletky = '171' THEN
                i:= 1;
            ELSIF PrecitaneCisloPaletky = '164' THEN
                i:= 2;
            ELSIF PrecitaneCisloPaletky = '181' THEN
                i:= 3;
            ELSIF PrecitaneCisloPaletky = '168' THEN
                i:= 4;
            ELSIF PrecitaneCisloPaletky = '140' THEN
                i:= 5;
            ELSIF PrecitaneCisloPaletky = '110' THEN
                i:= 6;
            ELSIF PrecitaneCisloPaletky = '156' THEN
                i:= 7;
            ELSIF PrecitaneCisloPaletky = '127' THEN
                i:= 8;
            ELSIF PrecitaneCisloPaletky = '139' THEN
                i:= 9;
            ELSIF PrecitaneCisloPaletky = '131' THEN
                i:= 10;
            ELSIF PrecitaneCisloPaletky = '178' THEN
                i:= 11;
            ELSIF PrecitaneCisloPaletky = '206' THEN
                i:= 12;
            ELSIF PrecitaneCisloPaletky = '119' THEN
                i:= 13;
            ELSIF PrecitaneCisloPaletky = '163' THEN
                i:= 14;
            ELSIF PrecitaneCisloPaletky = '128' THEN
                i:= 15;
            ELSIF PrecitaneCisloPaletky = '175' THEN
                i:= 16;
            ELSIF PrecitaneCisloPaletky = '138' THEN
                i:= 17;
            ELSE
                P34_Alarmy[429]:= TRUE;
                P4_PoruchaST2:= TRUE;
            END_IF

            IF i<> 0 THEN
                Paletka[i].PAR.CisloPaletky:= USINT_TO_STRING(i);
                PrecitaneCisloPaletky:= '';
                SC_P4_FunkcnyTestB.ResetStep:= TRUE;
                SC_P4_FunkcnyTestB.Step:= 103;
            END_IF

        103:
            SC_P4_FunkcnyTestB.StepName:='103 - Automaticky Rezim - kontrola stavu paletky';
            SC_P4_FunkcnyTestB.IdleTime.PT:= T#200ms;
            SC_P4_FunkcnyTestB.AlarmTime.PT:= T#5s;

            IF Paletka[i].PAR.TestovaciKus AND Paletka[i].PAR.CisloTestovacejStanice = 'ST_FT1,FT2' THEN
                IF P4_FunkcnyTestB.STAV.Tester_ON THEN
                    TestovaciKus:= TRUE;
                    SC_P4_FunkcnyTestB.ResetStep:= TRUE;
                    SC_P4_FunkcnyTestB.Step:= 118;
                ELSE
                    SC_P4_FunkcnyTestB.ResetStep:= TRUE;
                    SC_P4_FunkcnyTestB.Step:= 560;
                END_IF
            ELSIF Paletka[i].PAR.TestovaciKus AND Paletka[i].PAR.CisloTestovacejStanice <> 'ST_FT1,FT2' THEN
                SC_P4_FunkcnyTestB.ResetStep:= TRUE;
                SC_P4_FunkcnyTestB.Step:= 560;
            ELSIF Paletka[i].PAR.RevorkovyKus AND Paletka[i].PAR.CisloRevorkovejStanice = 'ST_FT1,FT2' THEN
                IF P4_FunkcnyTestB.STAV.Tester_ON THEN
                    Revork:= TRUE;
                    SC_P4_FunkcnyTestB.ResetStep:= TRUE;
                    SC_P4_FunkcnyTestB.Step:= 105;
                ELSE
                    SC_P4_FunkcnyTestB.ResetStep:= TRUE;
                    SC_P4_FunkcnyTestB.Step:= 560;
                END_IF
            ELSIF Paletka[i].PAR.RevorkovyKus AND Paletka[i].PAR.CisloRevorkovejStanice <> 'ST_FT1,FT2' THEN
                Revork:= FALSE;
                SC_P4_FunkcnyTestB.ResetStep:= TRUE;
                SC_P4_FunkcnyTestB.Step:= 560;
            ELSIF Paletka[i].PAR.StavPaletky = 'OK' AND P4_FunkcnyTestB.STAV.Tester_ON THEN
                SC_P4_FunkcnyTestB.ResetStep:= TRUE;
                SC_P4_FunkcnyTestB.Step:= 105;
            ELSIF Paletka[i].PAR.StavPaletky = 'OK' AND NOT P4_FunkcnyTestB.STAV.Tester_ON THEN
                SC_P4_FunkcnyTestB.ResetStep:= TRUE;
                SC_P4_FunkcnyTestB.Step:= 560;
            ELSIF Paletka[i].PAR.StavPaletky = 'NG' THEN
                SC_P4_FunkcnyTestB.ResetStep:= TRUE;
                SC_P4_FunkcnyTestB.Step:= 560;
            END_IF

        105:
            SC_P4_FunkcnyTestB.StepName:='105 - Automaticky Rezim - kontrola ukoncenia funkcneho testu';
            SC_P4_FunkcnyTestB.IdleTime.PT:= T#200ms;
            SC_P4_FunkcnyTestB.AlarmTime.PT:= T#5s;

            IF Paletka[i].VnutornyStav.FunkcnyTest_Ukonceny THEN
                SC_P4_FunkcnyTestB.ResetStep:= TRUE;
                SC_P4_FunkcnyTestB.Step:= 560;
            ELSE
                SC_P4_FunkcnyTestB.ResetStep:= TRUE;
                SC_P4_FunkcnyTestB.Step:= 110;
            END_IF

        110:
            SC_P4_FunkcnyTestB.StepName:='110 - Automaticky Rezim - cakam na prichod paletky na stanicu A a spustenie testovania';
            SC_P4_FunkcnyTestB.IdleTime.PT:= T#5s;
            SC_P4_FunkcnyTestB.AlarmTime.PT:= T#10s;
            SC_P4_FunkcnyTestB.AlarmTime.IN:= TRUE;

            IF NOT P3_LeakageTestA.IN.PritomnostPaletky_S23 AND
                NOT P3_LeakageTestB.IN.PritomnostPaletky_S24 AND
                NOT P4_FunkcnyTestA.IN.PritomnostPaletky_S10 THEN
                SC_P4_FunkcnyTestB.IdleTime.IN:= TRUE;
            ELSE
                SC_P4_FunkcnyTestB.IdleTime.IN:= FALSE;
            END_IF

            (*SC_P4_FunkcnyTestB.IdleTime.IN:= NOT P4_FunkcnyTestA.IN.PritomnostPaletky_S10;*)

            IF P4_FunkcnyTestB.KoniecCyklu THEN
                SC_P4_FunkcnyTestB.ResetStep:= TRUE;
                SC_P4_FunkcnyTestB.Step:= 118;
            ELSIF SC_P4_FunkcnyTestA.Step = 110 AND P4_FunkcnyTestA.IN.PritomnostPaletky_S10 THEN
                P4_FunkcnyTestB.OUT.KOM_StanicaA_StartTestovania:= TRUE;
                SC_P4_FunkcnyTestB.ResetStep:= TRUE;
                SC_P4_FunkcnyTestB.Step:= 118;
            ELSIF SC_P4_FunkcnyTestA.Step = 560 AND P4_FunkcnyTestA.IN.PritomnostPaletky_S10 THEN
                SC_P4_FunkcnyTestB.ResetStep:= TRUE;
                SC_P4_FunkcnyTestB.Step:= 118;
            ELSIF NOT P4_FunkcnyTestA.STAV.Tester_ON THEN
                SC_P4_FunkcnyTestB.ResetStep:= TRUE;
                SC_P4_FunkcnyTestB.Step:= 118;
            ELSIF SC_P4_FunkcnyTestB.IdleTime.Q THEN
                SC_P4_FunkcnyTestB.ResetStep:= TRUE;
                SC_P4_FunkcnyTestB.Step:= 118;
            ELSIF SC_P4_FunkcnyTestB.AlarmTime.Q THEN
                SC_P4_FunkcnyTestB.ResetStep:= TRUE;
                SC_P4_FunkcnyTestB.Step:= 118;
            END_IF

        118:
            SC_P4_FunkcnyTestB.StepName:='118 - Automaticky Rezim - zacentrovanie paletky';
            SC_P4_FunkcnyTestB.IdleTime.PT:= T#200ms;
            SC_P4_FunkcnyTestB.AlarmTime.PT:= T#5s;

            IF NOT SC_P4_FunkcnyTestB.Switch1 THEN
                Centrovacku_VYSUN:= TRUE;
                SC_P4_FunkcnyTestB.Switch1:= TRUE;
            END_IF

            IF P4_FunkcnyTestB.IN.Centrovanie_VYSUNUTE_MS30 THEN
                SC_P4_FunkcnyTestB.ResetStep:= TRUE;
                SC_P4_FunkcnyTestB.Step:= 120;
            END_IF

        120:
            SC_P4_FunkcnyTestB.StepName:='120 - Automaticky Rezim - zapnutie pruzenia vrchnych kontaktov';
            SC_P4_FunkcnyTestB.IdleTime.PT:= T#200ms;
            SC_P4_FunkcnyTestB.AlarmTime.PT:= T#5s;

            IF NOT SC_P4_FunkcnyTestB.Switch1 THEN
                P4_FunkcnyTestB.OUT.OdpruzenieKontaktov_VYPNI_YV188:= FALSE;
                P4_FunkcnyTestB.OUT.OdpruzenieKontaktov_ZAPNI_YV187:= TRUE;
                SC_P4_FunkcnyTestB.IdleTime.IN:= TRUE;
                SC_P4_FunkcnyTestB.Switch1:= TRUE;
            END_IF

            IF SC_P4_FunkcnyTestB.IdleTime.Q THEN
                SC_P4_FunkcnyTestB.ResetStep:= TRUE;
                SC_P4_FunkcnyTestB.Step:= 123;
            END_IF

        123:
            SC_P4_FunkcnyTestB.StepName:='123 - Automaticky Rezim - vysunutie hornych kontaktov';
            SC_P4_FunkcnyTestB.IdleTime.PT:= T#200ms;
            SC_P4_FunkcnyTestB.AlarmTime.PT:= T#5s;

            IF NOT SC_P4_FunkcnyTestB.Switch1 THEN
                HorneKontakty_VYSUN:= TRUE;
                SC_P4_FunkcnyTestB.Switch1:= TRUE;
            END_IF

            IF P4_FunkcnyTestB.IN.HorneKontakty_VYSUNUTE_MS26 THEN
                SC_P4_FunkcnyTestB.ResetStep:= TRUE;
                SC_P4_FunkcnyTestB.Step:= 125;
            END_IF

        125:
            SC_P4_FunkcnyTestB.StepName:='125 - Automaticky Rezim - vysunutie spodnych kontaktov';
            SC_P4_FunkcnyTestB.IdleTime.PT:= T#200ms;
            SC_P4_FunkcnyTestB.AlarmTime.PT:= T#5s;

            IF NOT SC_P4_FunkcnyTestB.Switch1 THEN
                SpodneKontakty_VYSUN:= TRUE;
                SC_P4_FunkcnyTestB.Switch1:= TRUE;
            END_IF

            IF P4_FunkcnyTestB.IN.SpodneKontakty_VYSUNUTE_MS34 THEN
                SC_P4_FunkcnyTestB.ResetStep:= TRUE;
                SC_P4_FunkcnyTestB.Step:= 127;
            END_IF

        127:
            SC_P4_FunkcnyTestB.StepName:='127 - Automaticky Rezim - pritlacenie kontaktov';
            SC_P4_FunkcnyTestB.IdleTime.PT:= T#200ms;
            SC_P4_FunkcnyTestB.AlarmTime.PT:= T#5s;

            IF Linka.PAR.ZvolenyModel = '4F' THEN
                P4_FunkcnyTestB.OUT.KontaktyTestera_VYSUN_YV172:= TRUE;
                SC_P4_FunkcnyTestB.IdleTime.IN:= TRUE;
            ELSIF Linka.PAR.ZvolenyModel = '5F' THEN
                P4_FunkcnyTestB.OUT.KontaktyTestera_VYSUN_YV172:= TRUE;
                SC_P4_FunkcnyTestB.IdleTime.IN:= TRUE;
            ELSIF Linka.PAR.ZvolenyModel = '5H' THEN
                SC_P4_FunkcnyTestB.ResetStep:= TRUE;
                SC_P4_FunkcnyTestB.Step:= 130;
            END_IF

            IF SC_P4_FunkcnyTestB.IdleTime.Q THEN
                SC_P4_FunkcnyTestB.ResetStep:= TRUE;
                SC_P4_FunkcnyTestB.Step:= 130;
            END_IF

        130:
            SC_P4_FunkcnyTestB.StepName:='130 - Automaticky Rezim - spustenie testovania';
            SC_P4_FunkcnyTestB.IdleTime.PT:= T#5s;
            SC_P4_FunkcnyTestB.AlarmTime.PT:= T#5s;

            IF NOT SC_P4_FunkcnyTestB.Switch1 THEN
                FV_Test_UKONCENY:= FALSE;
                FV_Test_START:= TRUE;
                SC_P4_FunkcnyTestB.Switch1:= TRUE;
            END_IF

            IF FV_Test_START AND FV_Test_UKONCENY THEN
                FV_Test_START:= FALSE;
                SC_P4_FunkcnyTestB.ResetStep:= TRUE;
                SC_P4_FunkcnyTestB.Step:= 140;
            END_IF

        140:
            SC_P4_FunkcnyTestB.StepName:='140 - Automaticky Rezim - vyhodnotenie testovania';
            SC_P4_FunkcnyTestB.IdleTime.PT:= T#200ms;
            SC_P4_FunkcnyTestB.AlarmTime.PT:= T#5s;

            IF P4_FunkcnyTestB.STAV.Vysledok_FV_Testu = 'OK' THEN
                Paletka[i].PAR.StavPowerCP:= 'PASS';
                Paletka[i].PAR.StavPaletky:= 'OK';
                Paletka[i].VnutornyStav.FunkcnyTest_Ukonceny:= TRUE;
                SC_P4_FunkcnyTestB.ResetStep:= TRUE;
                SC_P4_FunkcnyTestB.Step:= 145;
            ELSIF P4_FunkcnyTestB.STAV.Vysledok_FV_Testu = 'NG' THEN
                IF NOT Revork THEN
                    OpakovanyTest:= TRUE;
                END_IF
                Paletka[i].PAR.StavPowerCP:= 'FAIL';
                Paletka[i].PAR.StavPaletky:= 'NG';
                SC_P4_FunkcnyTestB.ResetStep:= TRUE;
                SC_P4_FunkcnyTestB.Step:= 145;
            END_IF

        145:
            SC_P4_FunkcnyTestB.StepName:='127 - Automaticky Rezim - vypnutie pritlacenie kontaktov';
            SC_P4_FunkcnyTestB.IdleTime.PT:= T#200ms;
            SC_P4_FunkcnyTestB.AlarmTime.PT:= T#5s;

            P4_FunkcnyTestB.OUT.KontaktyTestera_VYSUN_YV172:= FALSE;
            SC_P4_FunkcnyTestB.ResetStep:= TRUE;
            SC_P4_FunkcnyTestB.Step:= 148;

        148:
            SC_P4_FunkcnyTestB.StepName:='148 - Automaticky Rezim - zasunutie spodnych kontaktov';
            SC_P4_FunkcnyTestB.IdleTime.PT:= T#200ms;
            SC_P4_FunkcnyTestB.AlarmTime.PT:= T#5s;

            IF NOT SC_P4_FunkcnyTestB.Switch1 THEN
                SpodneKontakty_ZASUN:= TRUE;
                SC_P4_FunkcnyTestB.Switch1:= TRUE;
            END_IF

            IF P4_FunkcnyTestB.IN.SpodneKontakty_ZASUNUTE_MS32 THEN
                SC_P4_FunkcnyTestB.ResetStep:= TRUE;
                SC_P4_FunkcnyTestB.Step:= 150;
            END_IF

        150:
            SC_P4_FunkcnyTestB.StepName:='150 - Automaticky Rezim - zasunutie hornych kontaktov';
            SC_P4_FunkcnyTestB.IdleTime.PT:= T#200ms;
            SC_P4_FunkcnyTestB.AlarmTime.PT:= T#5s;

            IF NOT SC_P4_FunkcnyTestB.Switch1 THEN
                HorneKontakty_ZASUN:= TRUE;
                SC_P4_FunkcnyTestB.Switch1:= TRUE;
            END_IF

            IF P4_FunkcnyTestB.IN.HorneKontakty_ZASUNUTE_MS24 THEN
                SC_P4_FunkcnyTestB.ResetStep:= TRUE;
                SC_P4_FunkcnyTestB.Step:= 153;
            END_IF

        153:
            SC_P4_FunkcnyTestB.StepName:='153 - Automaticky Rezim - vypnutie pruzenia vrchnych kontaktov';
            SC_P4_FunkcnyTestB.IdleTime.PT:= T#200ms;
            SC_P4_FunkcnyTestB.AlarmTime.PT:= T#5s;

            IF NOT SC_P4_FunkcnyTestB.Switch1 THEN
                P4_FunkcnyTestB.OUT.OdpruzenieKontaktov_ZAPNI_YV187:= FALSE;
                P4_FunkcnyTestB.OUT.OdpruzenieKontaktov_VYPNI_YV188:= TRUE;
                SC_P4_FunkcnyTestB.IdleTime.IN:= TRUE;
                SC_P4_FunkcnyTestB.Switch1:= TRUE;
            END_IF

            IF SC_P4_FunkcnyTestB.IdleTime.Q THEN
                SC_P4_FunkcnyTestB.ResetStep:= TRUE;
                SC_P4_FunkcnyTestB.Step:= 545;
            END_IF

            //Odcentrovanie paletky//

        545:
            SC_P4_FunkcnyTestB.StepName:='545 - Automaticky Rezim - odcentrovanie paletky';
            SC_P4_FunkcnyTestB.IdleTime.PT:= T#200ms;
            SC_P4_FunkcnyTestB.AlarmTime.PT:= T#5s;

            IF NOT SC_P4_FunkcnyTestB.Switch1 THEN
                Centrovacku_ZASUN:= TRUE;
                SC_P4_FunkcnyTestB.Switch1:= TRUE;
            END_IF

            IF P4_FunkcnyTestB.IN.Centrovanie_ZASUNUTE_MS28 THEN
                SC_P4_FunkcnyTestB.ResetStep:= TRUE;
                SC_P4_FunkcnyTestB.Step:= 554;
            END_IF

        554:
            SC_P4_FunkcnyTestB.StepName:='554 - Automaticky Rezim - kontrola poctu testovani';
            SC_P4_FunkcnyTestB.IdleTime.PT:= T#1s;
            SC_P4_FunkcnyTestB.AlarmTime.PT:= T#5s;
            SC_P4_FunkcnyTestB.IdleTime.IN:= TRUE;

            IF NOT SC_P4_FunkcnyTestB.Switch1 THEN
                PocetOpakovaniTestu:= PocetOpakovaniTestu + 1;
                SC_P4_FunkcnyTestB.Switch1:= TRUE;
            END_IF

            IF OpakovanyTest AND PocetOpakovaniTestu < 2 AND SC_P4_FunkcnyTestB.IdleTime.Q AND NOT TestovaciKus THEN
                OpakovanyTest:= FALSE;
                SC_P4_FunkcnyTestB.ResetStep:= TRUE;
                SC_P4_FunkcnyTestB.Step:= 118;
            ELSIF OpakovanyTest AND PocetOpakovaniTestu >= 2 AND NOT TestovaciKus THEN
                Paletka[i].VnutornyStav.FunkcnyTest_Ukonceny:= TRUE;
                OpakovanyTest:= FALSE;
                PocetOpakovaniTestu:= 0;
                SC_P4_FunkcnyTestB.ResetStep:= TRUE;
                SC_P4_FunkcnyTestB.Step:= 555;
            ELSIF NOT OpakovanyTest OR TestovaciKus THEN
                SC_P4_FunkcnyTestB.ResetStep:= TRUE;
                SC_P4_FunkcnyTestB.Step:= 555;
            END_IF

        555:
            SC_P4_FunkcnyTestB.StepName:='555 - Automaticky Rezim - vyhodnotenie stavu paletky';
            SC_P4_FunkcnyTestB.IdleTime.PT:= T#200ms;
            SC_P4_FunkcnyTestB.AlarmTime.PT:= T#5s;

            IF Paletka[i].PAR.StavPaletky = 'OK' THEN
                IF Paletka[i].PAR.StavPowerCP = 'PASS' THEN
                    Paletka[i].PAR.StavPaletky:= 'OK';
                ELSIF Paletka[i].PAR.StavPowerCP = 'FAIL' THEN
                    Paletka[i].PAR.StavPaletky:= 'NG';
                END_IF
            END_IF

            SC_P4_FunkcnyTestB.ResetStep:= TRUE;
            SC_P4_FunkcnyTestB.Step:= 560;

            //Vyvezenie paletky//

        560:
            SC_P4_FunkcnyTestB.StepName:='560 - Automaticky Rezim - cakam na vyvezenie na stoper etiketovacky';
            SC_P4_FunkcnyTestB.IdleTime.PT:= T#200ms;
            SC_P4_FunkcnyTestB.AlarmTime.PT:= T#5s;

            IF P4_FunkcnyTestB.KoniecCyklu THEN
                SC_P4_FunkcnyTestB.ResetStep:= TRUE;
                SC_P4_FunkcnyTestB.Step:= 0;
            ELSIF (NOT P4_Etiketovacka.IN.PritomnostPaletky_S12 AND Safety.STAV.P4_VstupBunky_Bariera_AKTIVNA AND SC_P4_Etiketovacka.Step = 100) AND NOT P4_FunkcnyTestB.STAV.PrebiehaVyvezeniePaletky AND NOT TEST THEN
                P4_FunkcnyTestB.OUT.ZasunStoper_YV164:= TRUE;
                P4_FunkcnyTestB.STAV.PrebiehaVyvezeniePaletky:= TRUE;
                SC_P4_FunkcnyTestB.ResetStep:= TRUE;
                SC_P4_FunkcnyTestB.Step:= 561;
            END_IF

        561:
            SC_P4_FunkcnyTestB.StepName:='561 - Automaticky Rezim - ukoncenie vyvazania na stoper etiketovacky';
            SC_P4_FunkcnyTestB.IdleTime.PT:= T#200ms;
            SC_P4_FunkcnyTestB.AlarmTime.PT:= T#10s;

            SC_P4_FunkcnyTestB.IdleTime.IN:= NOT P4_FunkcnyTestB.IN.PritomnostPaletky_S11;
            SC_P4_FunkcnyTestB.AlarmTime.IN:= P4_FunkcnyTestB.IN.PritomnostPaletky_S11;

            IF NOT P4_FunkcnyTestB.IN.PritomnostPaletky_S11 THEN
                IF Revork THEN
                    Paletka[i].PAR.RevorkovyKus:= FALSE;
                    Paletka[i].PAR.CisloRevorkovejStanice:= '';
                    Revork:= FALSE;
                END_IF
                P4_FunkcnyTestB.OUT.ZasunStoper_YV164:= FALSE;
                TestovaciKus:= FALSE;
                OpakovanyTest:= FALSE;
                PocetOpakovaniTestu:= 0;
                Paletka[i].PAR.StavPowerCP:= '';
            END_IF

            IF SC_P4_FunkcnyTestB.IdleTime.Q AND NOT P4_FunkcnyTestB.OUT.ZasunStoper_YV164 THEN
                SC_P4_FunkcnyTestB.ResetStep:= TRUE;
                SC_P4_FunkcnyTestB.Step:= 100;
            ELSIF SC_P4_FunkcnyTestB.AlarmTime.Q THEN
                P34_Alarmy[451]:= TRUE;
                P4_Pracovisko.KoniecCyklu:= TRUE;
                SC_P4_FunkcnyTestB.ResetStep:= TRUE;
                SC_P4_FunkcnyTestB.Step:= 0;
            END_IF

            //*******************************************************Manuálny režim*******************************************************************************//
        700:
            SC_P4_FunkcnyTestB.StepName:='700 - Manualny Rezim';
            SC_P4_FunkcnyTestB.IdleTime.PT:= T#8s;
            SC_P4_FunkcnyTestB.AlarmTime.PT:= T#5s;

            //Ovládanie odpruženia kontaktov//
            IF P4_FunkcnyTestB.RR_ZapniOdpruzenieKontaktov THEN
                P4_FunkcnyTestB.OUT.OdpruzenieKontaktov_VYPNI_YV188:= FALSE;
                P4_FunkcnyTestB.OUT.OdpruzenieKontaktov_ZAPNI_YV187:= TRUE;
            ELSE
                P4_FunkcnyTestB.OUT.OdpruzenieKontaktov_ZAPNI_YV187:= FALSE;
                P4_FunkcnyTestB.OUT.OdpruzenieKontaktov_VYPNI_YV188:= TRUE;
            END_IF

            //Ovládanie vysunutia kontaktov testera//
            P4_FunkcnyTestB.OUT.KontaktyTestera_VYSUN_YV172:= P4_FunkcnyTestB.RR_VysunKontaktyTestera;

    END_CASE

END_PROGRAM

PROGRAM _EXIT
	(* Insert code here *)

END_PROGRAM
```

#### Variables.var - Local variables
```iecst
VAR
	SC_OvlCentrovacky : SequenceControlTyp;
	Centrovacku_VYSUN : BOOL;
	Centrovacku_ZASUN : BOOL;
	PrecitaneCisloPaletky : STRING[3];
	ServerOdpoved_StavPowerCP : STRING[5];
	i : USINT;
	SC_OvlSpodnychKontaktov : SequenceControlTyp;
	SpodneKontakty_VYSUN : BOOL;
	SpodneKontakty_ZASUN : BOOL;
	SC_OvlHornychKontaktov : SequenceControlTyp;
	HorneKontakty_VYSUN : BOOL;
	HorneKontakty_ZASUN : BOOL;
	SC_OvlTesteraFT : SequenceControlTyp;
	SKTcpClientTester_0 : SKTcpClientTester;
	dataStr : STRING[32];
	FV_Test_START : BOOL;
	FV_Test_UKONCENY : BOOL;
	TEST : BOOL;
	FV_Test_PocetDopytovTestera : USINT;
	TestovaciKus : BOOL;
	Revork : BOOL;
	PocetDopytovNaTester : USINT;
	CasTestovania : TON;
	NameranyCasTestovania : TIME;
	Triger_0 : BOOL;
	Triger_1 : BOOL;
	PocetOpakovaniTestu : USINT;
	OpakovanyTest : BOOL;
END_VAR
```

#### IOLinkKomunikacia.st
```iecst
ACTION IOLinkKomunikacia:

	//Snímač paletky//
	P4_FunkcnyTestB.IN.PritomnostPaletky_S11:= P4_FunkcnyTestB.PAR.SnimacPaletky_IOLinkInputs[1].0;
	P4_FunkcnyTestB.IN.PrecitaneCisloPaletky_S11:= P4_FunkcnyTestB.PAR.SnimacPaletky_IOLinkInputs[9];

END_ACTION
```

#### OvlCentrovacky.st
```iecst
ACTION OvlCentrovacky:

	//Volanie funkcie SequenceControl//
	SequenceControl(SC:= SC_OvlCentrovacky);

	CASE SC_OvlCentrovacky.Step OF

		0:
			SC_OvlCentrovacky.StepName:= '0 - Nulovanie';
			Centrovacku_VYSUN:= FALSE;
			Centrovacku_ZASUN:= FALSE;
//			P4_FunkcnyTestB.OUT.VysunCentrovanie_YV191:= FALSE;
//			P4_FunkcnyTestB.OUT.ZasunCentrovanie_YV192:= FALSE;

			IF SC_P4_FunkcnyTestB.Step <> 0 THEN
				SC_OvlCentrovacky.ResetStep:= TRUE;
				SC_OvlCentrovacky.Step:= 1;
			END_IF

		1:
			SC_OvlCentrovacky.StepName:= '1 - Rozhodnutie o cinnosti';
			IF Centrovacku_VYSUN THEN
				SC_OvlCentrovacky.Step:= 10;
			ELSIF Centrovacku_ZASUN THEN
				SC_OvlCentrovacky.Step:= 20;
			END_IF

		10:
			SC_OvlCentrovacky.StepName:= '10 - Vysunutie centrovacky';
			SC_OvlCentrovacky.IdleTime.PT:= T#3s;
			SC_OvlCentrovacky.AlarmTime.PT:= T#3s;

			IF P4_FunkcnyTestB.Automat THEN
				SC_OvlCentrovacky.AlarmTime.IN:= TRUE;
			ELSE
				SC_OvlCentrovacky.IdleTime.IN:= TRUE;
			END_IF

			IF NOT SC_OvlCentrovacky.Switch1 THEN
				P4_FunkcnyTestB.OUT.ZasunCentrovanie_YV192:= FALSE;
				P4_FunkcnyTestB.OUT.VysunCentrovanie_YV191:= TRUE;
				SC_OvlCentrovacky.Switch1:= TRUE;
			END_IF

			IF P4_FunkcnyTestB.IN.Centrovanie_VYSUNUTE_MS30 OR SC_OvlCentrovacky.IdleTime.Q THEN
				SC_OvlCentrovacky.ResetStep:= TRUE;
				SC_OvlCentrovacky.Step:= 0;
			ELSIF SC_OvlCentrovacky.AlarmTime.Q THEN
				P34_Alarmy[402]:= TRUE;
				P4_PoruchaST2:= TRUE;
			END_IF

		20:
			SC_OvlCentrovacky.StepName:= '20 - Zasunutie centrovacky';
			SC_OvlCentrovacky.IdleTime.PT:= T#3s;
			SC_OvlCentrovacky.AlarmTime.PT:= T#3s;

			IF P4_FunkcnyTestB.Automat THEN
				SC_OvlCentrovacky.AlarmTime.IN:= TRUE;
			ELSE
				SC_OvlCentrovacky.IdleTime.IN:= TRUE;
			END_IF

			IF NOT SC_OvlCentrovacky.Switch1 THEN
				P4_FunkcnyTestB.OUT.VysunCentrovanie_YV191:= FALSE;
				P4_FunkcnyTestB.OUT.ZasunCentrovanie_YV192:= TRUE;
				SC_OvlCentrovacky.Switch1:= TRUE;
			END_IF

			IF P4_FunkcnyTestB.IN.Centrovanie_ZASUNUTE_MS28 OR SC_OvlCentrovacky.IdleTime.Q THEN
				SC_OvlCentrovacky.ResetStep:= TRUE;
				SC_OvlCentrovacky.Step:= 0;
			ELSIF SC_OvlCentrovacky.AlarmTime.Q THEN
				P34_Alarmy[403]:= TRUE;
				P4_PoruchaST2:= TRUE;
			END_IF

	END_CASE

END_ACTION
```
